LIN {X -44.717, Y 73.793, Z 53.25, A 0, B 90, C 0, E1 0, E2 0, E3 0, E4 0} C_DIS
LIN {X -42.585, Y 75.218, Z 53.25, A 0, B 90, C 0, E1 0, E2 0, E3 0, E4 0} C_DIS
LIN {X -40.331, Y 76.441, Z 53.25, A 0, B 90, C 0, E1 0, E2 0, E3 0, E4 0} C_DIS
LIN {X -37.99, Y 77.489, Z 53.25, A 0, B 90, C 0, E1 0, E2 0, E3 0, E4 0} C_DIS
LIN {X -35.582, Y 78.373, Z 53.25, A 0, B 90, C 0, E1 0, E2 0, E3 0, E4 0} C_DIS
LIN {X -33.121, Y 79.096, Z 53.25, A 0, B 90, C 0, E1 0, E2 0, E3 0, E4 0} C_DIS
LIN {X -30.62, Y 79.664, Z 53.25, A 0, B 90, C 0, E1 0, E2 0, E3 0, E4 0} C_DIS
LIN {X -28.088, Y 80.079, Z 53.25, A 0, B 90, C 0, E1 0, E2 0, E3 0, E4 0} C_DIS
LIN {X -25.538, Y 80.347, Z 53.25, A 0, B 90, C 0, E1 0, E2 0, E3 0, E4 0} C_DIS
LIN {X -22.976, Y 80.479, Z 53.25, A 0, B 90, C 0, E1 0, E2 0, E3 0, E4 0} C_DIS
LIN {X -20.411, Y 80.492, Z 53.25, A 0, B 90, C 0, E1 0, E2 0, E3 0, E4 0} C_DIS
LIN {X -17.847, Y 80.414, Z 53.25, A 0, B 90, C 0, E1 0, E2 0, E3 0, E4 0} C_DIS
LIN {X -15.284, Y 80.286, Z 53.25, A 0, B 90, C 0, E1 0, E2 0, E3 0, E4 0} C_DIS
LIN {X -12.723, Y 80.139, Z 53.25, A 0, B 90, C 0, E1 0, E2 0, E3 0, E4 0} C_DIS
LIN {X -10.163, Y 79.971, Z 53.25, A 0, B 90, C 0, E1 0, E2 0, E3 0, E4 0} C_DIS
LIN {X -7.607, Y 79.756, Z 53.25, A 0, B 90, C 0, E1 0, E2 0, E3 0, E4 0} C_DIS
LIN {X -5.057, Y 79.475, Z 53.25, A 0, B 90, C 0, E1 0, E2 0, E3 0, E4 0} C_DIS
LIN {X -2.517, Y 79.116, Z 53.25, A 0, B 90, C 0, E1 0, E2 0, E3 0, E4 0} C_DIS
LIN {X 0, Y 78.658, Z 53.25, A 0, B 90, C 0, E1 0, E2 0, E3 0, E4 0} C_DIS
LIN {X 2.44, Y 77.975, Z 53.25, A 0, B 90, C 0, E1 0, E2 0, E3 0, E4 0} C_DIS
LIN {X 4.923, Y 77.332, Z 53.25, A 0, B 90, C 0, E1 0, E2 0, E3 0, E4 0} C_DIS
LIN {X 7.38, Y 76.595, Z 53.25, A 0, B 90, C 0, E1 0, E2 0, E3 0, E4 0} C_DIS
LIN {X 9.8, Y 75.743, Z 53.25, A 0, B 90, C 0, E1 0, E2 0, E3 0, E4 0} C_DIS
LIN {X 12.156, Y 74.73, Z 53.25, A 0, B 90, C 0, E1 0, E2 0, E3 0, E4 0} C_DIS
LIN {X 14.414, Y 73.515, Z 53.25, A 0, B 90, C 0, E1 0, E2 0, E3 0, E4 0} C_DIS
LIN {X 16.599, Y 72.171, Z 53.25, A 0, B 90, C 0, E1 0, E2 0, E3 0, E4 0} C_DIS
LIN {X 18.763, Y 70.793, Z 53.25, A 0, B 90, C 0, E1 0, E2 0, E3 0, E4 0} C_DIS
LIN {X 20.937, Y 69.431, Z 53.25, A 0, B 90, C 0, E1 0, E2 0, E3 0, E4 0} C_DIS
LIN {X 23.139, Y 68.116, Z 53.25, A 0, B 90, C 0, E1 0, E2 0, E3 0, E4 0} C_DIS
LIN {X 25.379, Y 66.866, Z 53.25, A 0, B 90, C 0, E1 0, E2 0, E3 0, E4 0} C_DIS
LIN {X 27.66, Y 65.691, Z 53.25, A 0, B 90, C 0, E1 0, E2 0, E3 0, E4 0} C_DIS
LIN {X 29.977, Y 64.59, Z 53.25, A 0, B 90, C 0, E1 0, E2 0, E3 0, E4 0} C_DIS
LIN {X 32.325, Y 63.556, Z 53.25, A 0, B 90, C 0, E1 0, E2 0, E3 0, E4 0} C_DIS
LIN {X 34.697, Y 62.581, Z 53.25, A 0, B 90, C 0, E1 0, E2 0, E3 0, E4 0} C_DIS
LIN {X 37.093, Y 61.664, Z 53.25, A 0, B 90, C 0, E1 0, E2 0, E3 0, E4 0} C_DIS
LIN {X 39.514, Y 60.816, Z 53.25, A 0, B 90, C 0, E1 0, E2 0, E3 0, E4 0} C_DIS
LIN {X 41.962, Y 60.049, Z 53.25, A 0, B 90, C 0, E1 0, E2 0, E3 0, E4 0} C_DIS
LIN {X 44.431, Y 59.352, Z 53.25, A 0, B 90, C 0, E1 0, E2 0, E3 0, E4 0} C_DIS
LIN {X 46.908, Y 58.684, Z 53.25, A 0, B 90, C 0, E1 0, E2 0, E3 0, E4 0} C_DIS
LIN {X 49.381, Y 58.001, Z 53.25, A 0, B 90, C 0, E1 0, E2 0, E3 0, E4 0} C_DIS
LIN {X 51.841, Y 57.274, Z 53.25, A 0, B 90, C 0, E1 0, E2 0, E3 0, E4 0} C_DIS
LIN {X 54.281, Y 56.483, Z 53.25, A 0, B 90, C 0, E1 0, E2 0, E3 0, E4 0} C_DIS
LIN {X 56.696, Y 55.617, Z 53.25, A 0, B 90, C 0, E1 0, E2 0, E3 0, E4 0} C_DIS
LIN {X 59.079, Y 54.667, Z 53.25, A 0, B 90, C 0, E1 0, E2 0, E3 0, E4 0} C_DIS
LIN {X 61.423, Y 53.627, Z 53.25, A 0, B 90, C 0, E1 0, E2 0, E3 0, E4 0} C_DIS
LIN {X 63.722, Y 52.488, Z 53.25, A 0, B 90, C 0, E1 0, E2 0, E3 0, E4 0} C_DIS
LIN {X 65.964, Y 51.243, Z 53.25, A 0, B 90, C 0, E1 0, E2 0, E3 0, E4 0} C_DIS
LIN {X 68.135, Y 49.877, Z 53.25, A 0, B 90, C 0, E1 0, E2 0, E3 0, E4 0} C_DIS
LIN {X 70.208, Y 48.366, Z 53.25, A 0, B 90, C 0, E1 0, E2 0, E3 0, E4 0} C_DIS
LIN {X 72.121, Y 46.659, Z 53.25, A 0, B 90, C 0, E1 0, E2 0, E3 0, E4 0} C_DIS
LIN {X 73.793, Y 44.717, Z 53.25, A 0, B 90, C 0, E1 0, E2 0, E3 0, E4 0} C_DIS
LIN {X 75.218, Y 42.585, Z 53.25, A 0, B 90, C 0, E1 0, E2 0, E3 0, E4 0} C_DIS
LIN {X 76.441, Y 40.331, Z 53.25, A 0, B 90, C 0, E1 0, E2 0, E3 0, E4 0} C_DIS
LIN {X 77.489, Y 37.99, Z 53.25, A 0, B 90, C 0, E1 0, E2 0, E3 0, E4 0} C_DIS
LIN {X 78.373, Y 35.582, Z 53.25, A 0, B 90, C 0, E1 0, E2 0, E3 0, E4 0} C_DIS
LIN {X 79.096, Y 33.121, Z 53.25, A 0, B 90, C 0, E1 0, E2 0, E3 0, E4 0} C_DIS
LIN {X 79.664, Y 30.62, Z 53.25, A 0, B 90, C 0, E1 0, E2 0, E3 0, E4 0} C_DIS
LIN {X 80.079, Y 28.088, Z 53.25, A 0, B 90, C 0, E1 0, E2 0, E3 0, E4 0} C_DIS
LIN {X 80.347, Y 25.538, Z 53.25, A 0, B 90, C 0, E1 0, E2 0, E3 0, E4 0} C_DIS
LIN {X 80.479, Y 22.976, Z 53.25, A 0, B 90, C 0, E1 0, E2 0, E3 0, E4 0} C_DIS
LIN {X 80.492, Y 20.411, Z 53.25, A 0, B 90, C 0, E1 0, E2 0, E3 0, E4 0} C_DIS
LIN {X 80.414, Y 17.847, Z 53.25, A 0, B 90, C 0, E1 0, E2 0, E3 0, E4 0} C_DIS
LIN {X 80.286, Y 15.284, Z 53.25, A 0, B 90, C 0, E1 0, E2 0, E3 0, E4 0} C_DIS
LIN {X 80.139, Y 12.723, Z 53.25, A 0, B 90, C 0, E1 0, E2 0, E3 0, E4 0} C_DIS
LIN {X 79.971, Y 10.163, Z 53.25, A 0, B 90, C 0, E1 0, E2 0, E3 0, E4 0} C_DIS
LIN {X 79.756, Y 7.607, Z 53.25, A 0, B 90, C 0, E1 0, E2 0, E3 0, E4 0} C_DIS
LIN {X 79.475, Y 5.057, Z 53.25, A 0, B 90, C 0, E1 0, E2 0, E3 0, E4 0} C_DIS
LIN {X 79.116, Y 2.517, Z 53.25, A 0, B 90, C 0, E1 0, E2 0, E3 0, E4 0} C_DIS
LIN {X 78.658, Y 0, Z 53.25, A 0, B 90, C 0, E1 0, E2 0, E3 0, E4 0} C_DIS
LIN {X 77.975, Y -2.44, Z 53.25, A 0, B 90, C 0, E1 0, E2 0, E3 0, E4 0} C_DIS
LIN {X 77.332, Y -4.923, Z 53.25, A 0, B 90, C 0, E1 0, E2 0, E3 0, E4 0} C_DIS
LIN {X 76.595, Y -7.38, Z 53.25, A 0, B 90, C 0, E1 0, E2 0, E3 0, E4 0} C_DIS
LIN {X 75.743, Y -9.8, Z 53.25, A 0, B 90, C 0, E1 0, E2 0, E3 0, E4 0} C_DIS
LIN {X 74.73, Y -12.156, Z 53.25, A 0, B 90, C 0, E1 0, E2 0, E3 0, E4 0} C_DIS
LIN {X 73.515, Y -14.414, Z 53.25, A 0, B 90, C 0, E1 0, E2 0, E3 0, E4 0} C_DIS
LIN {X 72.171, Y -16.599, Z 53.25, A 0, B 90, C 0, E1 0, E2 0, E3 0, E4 0} C_DIS
LIN {X 70.793, Y -18.763, Z 53.25, A 0, B 90, C 0, E1 0, E2 0, E3 0, E4 0} C_DIS
LIN {X 69.431, Y -20.937, Z 53.25, A 0, B 90, C 0, E1 0, E2 0, E3 0, E4 0} C_DIS
LIN {X 68.116, Y -23.139, Z 53.25, A 0, B 90, C 0, E1 0, E2 0, E3 0, E4 0} C_DIS
LIN {X 66.866, Y -25.379, Z 53.25, A 0, B 90, C 0, E1 0, E2 0, E3 0, E4 0} C_DIS
LIN {X 65.691, Y -27.66, Z 53.25, A 0, B 90, C 0, E1 0, E2 0, E3 0, E4 0} C_DIS
LIN {X 64.59, Y -29.977, Z 53.25, A 0, B 90, C 0, E1 0, E2 0, E3 0, E4 0} C_DIS
LIN {X 63.556, Y -32.325, Z 53.25, A 0, B 90, C 0, E1 0, E2 0, E3 0, E4 0} C_DIS
LIN {X 62.581, Y -34.697, Z 53.25, A 0, B 90, C 0, E1 0, E2 0, E3 0, E4 0} C_DIS
LIN {X 61.664, Y -37.093, Z 53.25, A 0, B 90, C 0, E1 0, E2 0, E3 0, E4 0} C_DIS
LIN {X 60.816, Y -39.514, Z 53.25, A 0, B 90, C 0, E1 0, E2 0, E3 0, E4 0} C_DIS
LIN {X 60.049, Y -41.962, Z 53.25, A 0, B 90, C 0, E1 0, E2 0, E3 0, E4 0} C_DIS
LIN {X 59.352, Y -44.431, Z 53.25, A 0, B 90, C 0, E1 0, E2 0, E3 0, E4 0} C_DIS
LIN {X 58.684, Y -46.908, Z 53.25, A 0, B 90, C 0, E1 0, E2 0, E3 0, E4 0} C_DIS
LIN {X 58.001, Y -49.381, Z 53.25, A 0, B 90, C 0, E1 0, E2 0, E3 0, E4 0} C_DIS
LIN {X 57.274, Y -51.841, Z 53.25, A 0, B 90, C 0, E1 0, E2 0, E3 0, E4 0} C_DIS
LIN {X 56.483, Y -54.281, Z 53.25, A 0, B 90, C 0, E1 0, E2 0, E3 0, E4 0} C_DIS
LIN {X 55.617, Y -56.696, Z 53.25, A 0, B 90, C 0, E1 0, E2 0, E3 0, E4 0} C_DIS
LIN {X 54.667, Y -59.079, Z 53.25, A 0, B 90, C 0, E1 0, E2 0, E3 0, E4 0} C_DIS
LIN {X 53.627, Y -61.423, Z 53.25, A 0, B 90, C 0, E1 0, E2 0, E3 0, E4 0} C_DIS
LIN {X 52.488, Y -63.722, Z 53.25, A 0, B 90, C 0, E1 0, E2 0, E3 0, E4 0} C_DIS
LIN {X 51.243, Y -65.964, Z 53.25, A 0, B 90, C 0, E1 0, E2 0, E3 0, E4 0} C_DIS
LIN {X 49.877, Y -68.135, Z 53.25, A 0, B 90, C 0, E1 0, E2 0, E3 0, E4 0} C_DIS
LIN {X 48.366, Y -70.208, Z 53.25, A 0, B 90, C 0, E1 0, E2 0, E3 0, E4 0} C_DIS
LIN {X 46.659, Y -72.121, Z 53.25, A 0, B 90, C 0, E1 0, E2 0, E3 0, E4 0} C_DIS
LIN {X 44.717, Y -73.793, Z 53.25, A 0, B 90, C 0, E1 0, E2 0, E3 0, E4 0} C_DIS
LIN {X 42.585, Y -75.218, Z 53.25, A 0, B 90, C 0, E1 0, E2 0, E3 0, E4 0} C_DIS
LIN {X 40.331, Y -76.441, Z 53.25, A 0, B 90, C 0, E1 0, E2 0, E3 0, E4 0} C_DIS
LIN {X 37.99, Y -77.489, Z 53.25, A 0, B 90, C 0, E1 0, E2 0, E3 0, E4 0} C_DIS
LIN {X 35.582, Y -78.373, Z 53.25, A 0, B 90, C 0, E1 0, E2 0, E3 0, E4 0} C_DIS
LIN {X 33.121, Y -79.096, Z 53.25, A 0, B 90, C 0, E1 0, E2 0, E3 0, E4 0} C_DIS
LIN {X 30.62, Y -79.664, Z 53.25, A 0, B 90, C 0, E1 0, E2 0, E3 0, E4 0} C_DIS
LIN {X 28.088, Y -80.079, Z 53.25, A 0, B 90, C 0, E1 0, E2 0, E3 0, E4 0} C_DIS
LIN {X 25.538, Y -80.347, Z 53.25, A 0, B 90, C 0, E1 0, E2 0, E3 0, E4 0} C_DIS
LIN {X 22.976, Y -80.479, Z 53.25, A 0, B 90, C 0, E1 0, E2 0, E3 0, E4 0} C_DIS
LIN {X 20.411, Y -80.492, Z 53.25, A 0, B 90, C 0, E1 0, E2 0, E3 0, E4 0} C_DIS
LIN {X 17.847, Y -80.414, Z 53.25, A 0, B 90, C 0, E1 0, E2 0, E3 0, E4 0} C_DIS
LIN {X 15.284, Y -80.286, Z 53.25, A 0, B 90, C 0, E1 0, E2 0, E3 0, E4 0} C_DIS
LIN {X 12.723, Y -80.139, Z 53.25, A 0, B 90, C 0, E1 0, E2 0, E3 0, E4 0} C_DIS
LIN {X 10.163, Y -79.971, Z 53.25, A 0, B 90, C 0, E1 0, E2 0, E3 0, E4 0} C_DIS
LIN {X 7.607, Y -79.756, Z 53.25, A 0, B 90, C 0, E1 0, E2 0, E3 0, E4 0} C_DIS
LIN {X 5.057, Y -79.475, Z 53.25, A 0, B 90, C 0, E1 0, E2 0, E3 0, E4 0} C_DIS
LIN {X 2.517, Y -79.116, Z 53.25, A 0, B 90, C 0, E1 0, E2 0, E3 0, E4 0} C_DIS
LIN {X 0, Y -78.658, Z 53.25, A 0, B 90, C 0, E1 0, E2 0, E3 0, E4 0} C_DIS
LIN {X -2.44, Y -77.975, Z 53.25, A 0, B 90, C 0, E1 0, E2 0, E3 0, E4 0} C_DIS
LIN {X -4.923, Y -77.332, Z 53.25, A 0, B 90, C 0, E1 0, E2 0, E3 0, E4 0} C_DIS
LIN {X -7.38, Y -76.595, Z 53.25, A 0, B 90, C 0, E1 0, E2 0, E3 0, E4 0} C_DIS
LIN {X -9.8, Y -75.743, Z 53.25, A 0, B 90, C 0, E1 0, E2 0, E3 0, E4 0} C_DIS
LIN {X -12.156, Y -74.73, Z 53.25, A 0, B 90, C 0, E1 0, E2 0, E3 0, E4 0} C_DIS
LIN {X -14.414, Y -73.515, Z 53.25, A 0, B 90, C 0, E1 0, E2 0, E3 0, E4 0} C_DIS
LIN {X -16.599, Y -72.171, Z 53.25, A 0, B 90, C 0, E1 0, E2 0, E3 0, E4 0} C_DIS
LIN {X -18.763, Y -70.793, Z 53.25, A 0, B 90, C 0, E1 0, E2 0, E3 0, E4 0} C_DIS
LIN {X -20.937, Y -69.431, Z 53.25, A 0, B 90, C 0, E1 0, E2 0, E3 0, E4 0} C_DIS
LIN {X -23.139, Y -68.116, Z 53.25, A 0, B 90, C 0, E1 0, E2 0, E3 0, E4 0} C_DIS
LIN {X -25.379, Y -66.866, Z 53.25, A 0, B 90, C 0, E1 0, E2 0, E3 0, E4 0} C_DIS
LIN {X -27.66, Y -65.691, Z 53.25, A 0, B 90, C 0, E1 0, E2 0, E3 0, E4 0} C_DIS
LIN {X -29.977, Y -64.59, Z 53.25, A 0, B 90, C 0, E1 0, E2 0, E3 0, E4 0} C_DIS
LIN {X -32.325, Y -63.556, Z 53.25, A 0, B 90, C 0, E1 0, E2 0, E3 0, E4 0} C_DIS
LIN {X -34.697, Y -62.581, Z 53.25, A 0, B 90, C 0, E1 0, E2 0, E3 0, E4 0} C_DIS
LIN {X -37.093, Y -61.664, Z 53.25, A 0, B 90, C 0, E1 0, E2 0, E3 0, E4 0} C_DIS
LIN {X -39.514, Y -60.816, Z 53.25, A 0, B 90, C 0, E1 0, E2 0, E3 0, E4 0} C_DIS
LIN {X -41.962, Y -60.049, Z 53.25, A 0, B 90, C 0, E1 0, E2 0, E3 0, E4 0} C_DIS
LIN {X -44.431, Y -59.352, Z 53.25, A 0, B 90, C 0, E1 0, E2 0, E3 0, E4 0} C_DIS
LIN {X -46.908, Y -58.684, Z 53.25, A 0, B 90, C 0, E1 0, E2 0, E3 0, E4 0} C_DIS
LIN {X -49.381, Y -58.001, Z 53.25, A 0, B 90, C 0, E1 0, E2 0, E3 0, E4 0} C_DIS
LIN {X -51.841, Y -57.274, Z 53.25, A 0, B 90, C 0, E1 0, E2 0, E3 0, E4 0} C_DIS
LIN {X -54.281, Y -56.483, Z 53.25, A 0, B 90, C 0, E1 0, E2 0, E3 0, E4 0} C_DIS
LIN {X -56.696, Y -55.617, Z 53.25, A 0, B 90, C 0, E1 0, E2 0, E3 0, E4 0} C_DIS
LIN {X -59.079, Y -54.667, Z 53.25, A 0, B 90, C 0, E1 0, E2 0, E3 0, E4 0} C_DIS
LIN {X -61.423, Y -53.627, Z 53.25, A 0, B 90, C 0, E1 0, E2 0, E3 0, E4 0} C_DIS
LIN {X -63.722, Y -52.488, Z 53.25, A 0, B 90, C 0, E1 0, E2 0, E3 0, E4 0} C_DIS
LIN {X -65.964, Y -51.243, Z 53.25, A 0, B 90, C 0, E1 0, E2 0, E3 0, E4 0} C_DIS
LIN {X -68.135, Y -49.877, Z 53.25, A 0, B 90, C 0, E1 0, E2 0, E3 0, E4 0} C_DIS
LIN {X -70.208, Y -48.366, Z 53.25, A 0, B 90, C 0, E1 0, E2 0, E3 0, E4 0} C_DIS
LIN {X -72.121, Y -46.659, Z 53.25, A 0, B 90, C 0, E1 0, E2 0, E3 0, E4 0} C_DIS
LIN {X -73.793, Y -44.717, Z 53.25, A 0, B 90, C 0, E1 0, E2 0, E3 0, E4 0} C_DIS
LIN {X -75.218, Y -42.585, Z 53.25, A 0, B 90, C 0, E1 0, E2 0, E3 0, E4 0} C_DIS
LIN {X -76.441, Y -40.331, Z 53.25, A 0, B 90, C 0, E1 0, E2 0, E3 0, E4 0} C_DIS
LIN {X -77.489, Y -37.99, Z 53.25, A 0, B 90, C 0, E1 0, E2 0, E3 0, E4 0} C_DIS
LIN {X -78.373, Y -35.582, Z 53.25, A 0, B 90, C 0, E1 0, E2 0, E3 0, E4 0} C_DIS
LIN {X -79.096, Y -33.121, Z 53.25, A 0, B 90, C 0, E1 0, E2 0, E3 0, E4 0} C_DIS
LIN {X -79.664, Y -30.62, Z 53.25, A 0, B 90, C 0, E1 0, E2 0, E3 0, E4 0} C_DIS
LIN {X -80.079, Y -28.088, Z 53.25, A 0, B 90, C 0, E1 0, E2 0, E3 0, E4 0} C_DIS
LIN {X -80.347, Y -25.538, Z 53.25, A 0, B 90, C 0, E1 0, E2 0, E3 0, E4 0} C_DIS
LIN {X -80.479, Y -22.976, Z 53.25, A 0, B 90, C 0, E1 0, E2 0, E3 0, E4 0} C_DIS
LIN {X -80.492, Y -20.411, Z 53.25, A 0, B 90, C 0, E1 0, E2 0, E3 0, E4 0} C_DIS
LIN {X -80.414, Y -17.847, Z 53.25, A 0, B 90, C 0, E1 0, E2 0, E3 0, E4 0} C_DIS
LIN {X -80.286, Y -15.284, Z 53.25, A 0, B 90, C 0, E1 0, E2 0, E3 0, E4 0} C_DIS
LIN {X -80.139, Y -12.723, Z 53.25, A 0, B 90, C 0, E1 0, E2 0, E3 0, E4 0} C_DIS
LIN {X -79.971, Y -10.163, Z 53.25, A 0, B 90, C 0, E1 0, E2 0, E3 0, E4 0} C_DIS
LIN {X -79.756, Y -7.607, Z 53.25, A 0, B 90, C 0, E1 0, E2 0, E3 0, E4 0} C_DIS
LIN {X -79.475, Y -5.057, Z 53.25, A 0, B 90, C 0, E1 0, E2 0, E3 0, E4 0} C_DIS
LIN {X -79.116, Y -2.517, Z 53.25, A 0, B 90, C 0, E1 0, E2 0, E3 0, E4 0} C_DIS
LIN {X -78.665, Y 0, Z 55.75, A 0, B 90, C 0, E1 0, E2 0, E3 0, E4 0} C_DIS
LIN {X -77.946, Y 2.433, Z 55.75, A 0, B 90, C 0, E1 0, E2 0, E3 0, E4 0} C_DIS
LIN {X -77.272, Y 4.917, Z 55.75, A 0, B 90, C 0, E1 0, E2 0, E3 0, E4 0} C_DIS
LIN {X -76.503, Y 7.373, Z 55.75, A 0, B 90, C 0, E1 0, E2 0, E3 0, E4 0} C_DIS
LIN {X -75.619, Y 9.789, Z 55.75, A 0, B 90, C 0, E1 0, E2 0, E3 0, E4 0} C_DIS
LIN {X -74.571, Y 12.139, Z 55.75, A 0, B 90, C 0, E1 0, E2 0, E3 0, E4 0} C_DIS
LIN {X -73.32, Y 14.387, Z 55.75, A 0, B 90, C 0, E1 0, E2 0, E3 0, E4 0} C_DIS
LIN {X -71.942, Y 16.56, Z 55.75, A 0, B 90, C 0, E1 0, E2 0, E3 0, E4 0} C_DIS
LIN {X -70.532, Y 18.714, Z 55.75, A 0, B 90, C 0, E1 0, E2 0, E3 0, E4 0} C_DIS
LIN {X -69.142, Y 20.88, Z 55.75, A 0, B 90, C 0, E1 0, E2 0, E3 0, E4 0} C_DIS
LIN {X -67.803, Y 23.077, Z 55.75, A 0, B 90, C 0, E1 0, E2 0, E3 0, E4 0} C_DIS
LIN {X -66.534, Y 25.317, Z 55.75, A 0, B 90, C 0, E1 0, E2 0, E3 0, E4 0} C_DIS
LIN {X -65.347, Y 27.6, Z 55.75, A 0, B 90, C 0, E1 0, E2 0, E3 0, E4 0} C_DIS
LIN {X -64.241, Y 29.923, Z 55.75, A 0, B 90, C 0, E1 0, E2 0, E3 0, E4 0} C_DIS
LIN {X -63.207, Y 32.28, Z 55.75, A 0, B 90, C 0, E1 0, E2 0, E3 0, E4 0} C_DIS
LIN {X -62.239, Y 34.665, Z 55.75, A 0, B 90, C 0, E1 0, E2 0, E3 0, E4 0} C_DIS
LIN {X -61.336, Y 37.075, Z 55.75, A 0, B 90, C 0, E1 0, E2 0, E3 0, E4 0} C_DIS
LIN {X -60.509, Y 39.512, Z 55.75, A 0, B 90, C 0, E1 0, E2 0, E3 0, E4 0} C_DIS
LIN {X -59.769, Y 41.976, Z 55.75, A 0, B 90, C 0, E1 0, E2 0, E3 0, E4 0} C_DIS
LIN {X -59.105, Y 44.463, Z 55.75, A 0, B 90, C 0, E1 0, E2 0, E3 0, E4 0} C_DIS
LIN {X -58.473, Y 46.958, Z 55.75, A 0, B 90, C 0, E1 0, E2 0, E3 0, E4 0} C_DIS
LIN {X -57.827, Y 49.449, Z 55.75, A 0, B 90, C 0, E1 0, E2 0, E3 0, E4 0} C_DIS
LIN {X -57.137, Y 51.928, Z 55.75, A 0, B 90, C 0, E1 0, E2 0, E3 0, E4 0} C_DIS
LIN {X -56.382, Y 54.389, Z 55.75, A 0, B 90, C 0, E1 0, E2 0, E3 0, E4 0} C_DIS
LIN {X -55.552, Y 56.824, Z 55.75, A 0, B 90, C 0, E1 0, E2 0, E3 0, E4 0} C_DIS
LIN {X -54.636, Y 59.23, Z 55.75, A 0, B 90, C 0, E1 0, E2 0, E3 0, E4 0} C_DIS
LIN {X -53.628, Y 61.597, Z 55.75, A 0, B 90, C 0, E1 0, E2 0, E3 0, E4 0} C_DIS
LIN {X -52.52, Y 63.92, Z 55.75, A 0, B 90, C 0, E1 0, E2 0, E3 0, E4 0} C_DIS
LIN {X -51.303, Y 66.188, Z 55.75, A 0, B 90, C 0, E1 0, E2 0, E3 0, E4 0} C_DIS
LIN {X -49.964, Y 68.385, Z 55.75, A 0, B 90, C 0, E1 0, E2 0, E3 0, E4 0} C_DIS
LIN {X -48.475, Y 70.483, Z 55.75, A 0, B 90, C 0, E1 0, E2 0, E3 0, E4 0} C_DIS
LIN {X -46.785, Y 72.422, Z 55.75, A 0, B 90, C 0, E1 0, E2 0, E3 0, E4 0} C_DIS
LIN {X -44.848, Y 74.114, Z 55.75, A 0, B 90, C 0, E1 0, E2 0, E3 0, E4 0} C_DIS
LIN {X -42.715, Y 75.551, Z 55.75, A 0, B 90, C 0, E1 0, E2 0, E3 0, E4 0} C_DIS
LIN {X -40.455, Y 76.78, Z 55.75, A 0, B 90, C 0, E1 0, E2 0, E3 0, E4 0} C_DIS
LIN {X -38.105, Y 77.829, Z 55.75, A 0, B 90, C 0, E1 0, E2 0, E3 0, E4 0} C_DIS
LIN {X -35.687, Y 78.708, Z 55.75, A 0, B 90, C 0, E1 0, E2 0, E3 0, E4 0} C_DIS
LIN {X -33.215, Y 79.424, Z 55.75, A 0, B 90, C 0, E1 0, E2 0, E3 0, E4 0} C_DIS
LIN {X -30.703, Y 79.98, Z 55.75, A 0, B 90, C 0, E1 0, E2 0, E3 0, E4 0} C_DIS
LIN {X -28.161, Y 80.379, Z 55.75, A 0, B 90, C 0, E1 0, E2 0, E3 0, E4 0} C_DIS
LIN {X -25.599, Y 80.627, Z 55.75, A 0, B 90, C 0, E1 0, E2 0, E3 0, E4 0} C_DIS
LIN {X -23.028, Y 80.736, Z 55.75, A 0, B 90, C 0, E1 0, E2 0, E3 0, E4 0} C_DIS
LIN {X -20.455, Y 80.723, Z 55.75, A 0, B 90, C 0, E1 0, E2 0, E3 0, E4 0} C_DIS
LIN {X -17.884, Y 80.617, Z 55.75, A 0, B 90, C 0, E1 0, E2 0, E3 0, E4 0} C_DIS
LIN {X -15.315, Y 80.46, Z 55.75, A 0, B 90, C 0, E1 0, E2 0, E3 0, E4 0} C_DIS
LIN {X -12.747, Y 80.284, Z 55.75, A 0, B 90, C 0, E1 0, E2 0, E3 0, E4 0} C_DIS
LIN {X -10.181, Y 80.089, Z 55.75, A 0, B 90, C 0, E1 0, E2 0, E3 0, E4 0} C_DIS
LIN {X -7.619, Y 79.847, Z 55.75, A 0, B 90, C 0, E1 0, E2 0, E3 0, E4 0} C_DIS
LIN {X -5.064, Y 79.539, Z 55.75, A 0, B 90, C 0, E1 0, E2 0, E3 0, E4 0} C_DIS
LIN {X -2.52, Y 79.152, Z 55.75, A 0, B 90, C 0, E1 0, E2 0, E3 0, E4 0} C_DIS
LIN {X 0, Y 78.665, Z 55.75, A 0, B 90, C 0, E1 0, E2 0, E3 0, E4 0} C_DIS
LIN {X 2.433, Y 77.946, Z 55.75, A 0, B 90, C 0, E1 0, E2 0, E3 0, E4 0} C_DIS
LIN {X 4.917, Y 77.272, Z 55.75, A 0, B 90, C 0, E1 0, E2 0, E3 0, E4 0} C_DIS
LIN {X 7.373, Y 76.503, Z 55.75, A 0, B 90, C 0, E1 0, E2 0, E3 0, E4 0} C_DIS
LIN {X 9.789, Y 75.619, Z 55.75, A 0, B 90, C 0, E1 0, E2 0, E3 0, E4 0} C_DIS
LIN {X 12.139, Y 74.571, Z 55.75, A 0, B 90, C 0, E1 0, E2 0, E3 0, E4 0} C_DIS
LIN {X 14.387, Y 73.32, Z 55.75, A 0, B 90, C 0, E1 0, E2 0, E3 0, E4 0} C_DIS
LIN {X 16.56, Y 71.942, Z 55.75, A 0, B 90, C 0, E1 0, E2 0, E3 0, E4 0} C_DIS
LIN {X 18.714, Y 70.532, Z 55.75, A 0, B 90, C 0, E1 0, E2 0, E3 0, E4 0} C_DIS
LIN {X 20.88, Y 69.142, Z 55.75, A 0, B 90, C 0, E1 0, E2 0, E3 0, E4 0} C_DIS
LIN {X 23.077, Y 67.803, Z 55.75, A 0, B 90, C 0, E1 0, E2 0, E3 0, E4 0} C_DIS
LIN {X 25.317, Y 66.534, Z 55.75, A 0, B 90, C 0, E1 0, E2 0, E3 0, E4 0} C_DIS
LIN {X 27.6, Y 65.347, Z 55.75, A 0, B 90, C 0, E1 0, E2 0, E3 0, E4 0} C_DIS
LIN {X 29.923, Y 64.241, Z 55.75, A 0, B 90, C 0, E1 0, E2 0, E3 0, E4 0} C_DIS
LIN {X 32.28, Y 63.207, Z 55.75, A 0, B 90, C 0, E1 0, E2 0, E3 0, E4 0} C_DIS
LIN {X 34.665, Y 62.239, Z 55.75, A 0, B 90, C 0, E1 0, E2 0, E3 0, E4 0} C_DIS
LIN {X 37.075, Y 61.336, Z 55.75, A 0, B 90, C 0, E1 0, E2 0, E3 0, E4 0} C_DIS
LIN {X 39.512, Y 60.509, Z 55.75, A 0, B 90, C 0, E1 0, E2 0, E3 0, E4 0} C_DIS
LIN {X 41.976, Y 59.769, Z 55.75, A 0, B 90, C 0, E1 0, E2 0, E3 0, E4 0} C_DIS
LIN {X 44.463, Y 59.105, Z 55.75, A 0, B 90, C 0, E1 0, E2 0, E3 0, E4 0} C_DIS
LIN {X 46.958, Y 58.473, Z 55.75, A 0, B 90, C 0, E1 0, E2 0, E3 0, E4 0} C_DIS
LIN {X 49.449, Y 57.827, Z 55.75, A 0, B 90, C 0, E1 0, E2 0, E3 0, E4 0} C_DIS
LIN {X 51.928, Y 57.137, Z 55.75, A 0, B 90, C 0, E1 0, E2 0, E3 0, E4 0} C_DIS
LIN {X 54.389, Y 56.382, Z 55.75, A 0, B 90, C 0, E1 0, E2 0, E3 0, E4 0} C_DIS
LIN {X 56.824, Y 55.552, Z 55.75, A 0, B 90, C 0, E1 0, E2 0, E3 0, E4 0} C_DIS
LIN {X 59.23, Y 54.636, Z 55.75, A 0, B 90, C 0, E1 0, E2 0, E3 0, E4 0} C_DIS
LIN {X 61.597, Y 53.628, Z 55.75, A 0, B 90, C 0, E1 0, E2 0, E3 0, E4 0} C_DIS
LIN {X 63.92, Y 52.52, Z 55.75, A 0, B 90, C 0, E1 0, E2 0, E3 0, E4 0} C_DIS
LIN {X 66.188, Y 51.303, Z 55.75, A 0, B 90, C 0, E1 0, E2 0, E3 0, E4 0} C_DIS
LIN {X 68.385, Y 49.964, Z 55.75, A 0, B 90, C 0, E1 0, E2 0, E3 0, E4 0} C_DIS
LIN {X 70.483, Y 48.475, Z 55.75, A 0, B 90, C 0, E1 0, E2 0, E3 0, E4 0} C_DIS
LIN {X 72.422, Y 46.785, Z 55.75, A 0, B 90, C 0, E1 0, E2 0, E3 0, E4 0} C_DIS
LIN {X 74.114, Y 44.848, Z 55.75, A 0, B 90, C 0, E1 0, E2 0, E3 0, E4 0} C_DIS
LIN {X 75.551, Y 42.715, Z 55.75, A 0, B 90, C 0, E1 0, E2 0, E3 0, E4 0} C_DIS
LIN {X 76.78, Y 40.455, Z 55.75, A 0, B 90, C 0, E1 0, E2 0, E3 0, E4 0} C_DIS
LIN {X 77.829, Y 38.105, Z 55.75, A 0, B 90, C 0, E1 0, E2 0, E3 0, E4 0} C_DIS
LIN {X 78.708, Y 35.687, Z 55.75, A 0, B 90, C 0, E1 0, E2 0, E3 0, E4 0} C_DIS
LIN {X 79.424, Y 33.215, Z 55.75, A 0, B 90, C 0, E1 0, E2 0, E3 0, E4 0} C_DIS
LIN {X 79.98, Y 30.703, Z 55.75, A 0, B 90, C 0, E1 0, E2 0, E3 0, E4 0} C_DIS
LIN {X 80.379, Y 28.161, Z 55.75, A 0, B 90, C 0, E1 0, E2 0, E3 0, E4 0} C_DIS
LIN {X 80.627, Y 25.599, Z 55.75, A 0, B 90, C 0, E1 0, E2 0, E3 0, E4 0} C_DIS
LIN {X 80.736, Y 23.028, Z 55.75, A 0, B 90, C 0, E1 0, E2 0, E3 0, E4 0} C_DIS
LIN {X 80.723, Y 20.455, Z 55.75, A 0, B 90, C 0, E1 0, E2 0, E3 0, E4 0} C_DIS
LIN {X 80.617, Y 17.884, Z 55.75, A 0, B 90, C 0, E1 0, E2 0, E3 0, E4 0} C_DIS
LIN {X 80.46, Y 15.315, Z 55.75, A 0, B 90, C 0, E1 0, E2 0, E3 0, E4 0} C_DIS
LIN {X 80.284, Y 12.747, Z 55.75, A 0, B 90, C 0, E1 0, E2 0, E3 0, E4 0} C_DIS
LIN {X 80.089, Y 10.181, Z 55.75, A 0, B 90, C 0, E1 0, E2 0, E3 0, E4 0} C_DIS
LIN {X 79.847, Y 7.619, Z 55.75, A 0, B 90, C 0, E1 0, E2 0, E3 0, E4 0} C_DIS
LIN {X 79.539, Y 5.064, Z 55.75, A 0, B 90, C 0, E1 0, E2 0, E3 0, E4 0} C_DIS
LIN {X 79.152, Y 2.52, Z 55.75, A 0, B 90, C 0, E1 0, E2 0, E3 0, E4 0} C_DIS
LIN {X 78.665, Y 0, Z 55.75, A 0, B 90, C 0, E1 0, E2 0, E3 0, E4 0} C_DIS
LIN {X 77.946, Y -2.433, Z 55.75, A 0, B 90, C 0, E1 0, E2 0, E3 0, E4 0} C_DIS
LIN {X 77.272, Y -4.917, Z 55.75, A 0, B 90, C 0, E1 0, E2 0, E3 0, E4 0} C_DIS
LIN {X 76.503, Y -7.373, Z 55.75, A 0, B 90, C 0, E1 0, E2 0, E3 0, E4 0} C_DIS
LIN {X 75.619, Y -9.789, Z 55.75, A 0, B 90, C 0, E1 0, E2 0, E3 0, E4 0} C_DIS
LIN {X 74.571, Y -12.139, Z 55.75, A 0, B 90, C 0, E1 0, E2 0, E3 0, E4 0} C_DIS
LIN {X 73.32, Y -14.387, Z 55.75, A 0, B 90, C 0, E1 0, E2 0, E3 0, E4 0} C_DIS
LIN {X 71.942, Y -16.56, Z 55.75, A 0, B 90, C 0, E1 0, E2 0, E3 0, E4 0} C_DIS
LIN {X 70.532, Y -18.714, Z 55.75, A 0, B 90, C 0, E1 0, E2 0, E3 0, E4 0} C_DIS
LIN {X 69.142, Y -20.88, Z 55.75, A 0, B 90, C 0, E1 0, E2 0, E3 0, E4 0} C_DIS
LIN {X 67.803, Y -23.077, Z 55.75, A 0, B 90, C 0, E1 0, E2 0, E3 0, E4 0} C_DIS
LIN {X 66.534, Y -25.317, Z 55.75, A 0, B 90, C 0, E1 0, E2 0, E3 0, E4 0} C_DIS
LIN {X 65.347, Y -27.6, Z 55.75, A 0, B 90, C 0, E1 0, E2 0, E3 0, E4 0} C_DIS
LIN {X 64.241, Y -29.923, Z 55.75, A 0, B 90, C 0, E1 0, E2 0, E3 0, E4 0} C_DIS
LIN {X 63.207, Y -32.28, Z 55.75, A 0, B 90, C 0, E1 0, E2 0, E3 0, E4 0} C_DIS
LIN {X 62.239, Y -34.665, Z 55.75, A 0, B 90, C 0, E1 0, E2 0, E3 0, E4 0} C_DIS
LIN {X 61.336, Y -37.075, Z 55.75, A 0, B 90, C 0, E1 0, E2 0, E3 0, E4 0} C_DIS
LIN {X 60.509, Y -39.512, Z 55.75, A 0, B 90, C 0, E1 0, E2 0, E3 0, E4 0} C_DIS
LIN {X 59.769, Y -41.976, Z 55.75, A 0, B 90, C 0, E1 0, E2 0, E3 0, E4 0} C_DIS
LIN {X 59.105, Y -44.463, Z 55.75, A 0, B 90, C 0, E1 0, E2 0, E3 0, E4 0} C_DIS
LIN {X 58.473, Y -46.958, Z 55.75, A 0, B 90, C 0, E1 0, E2 0, E3 0, E4 0} C_DIS
LIN {X 57.827, Y -49.449, Z 55.75, A 0, B 90, C 0, E1 0, E2 0, E3 0, E4 0} C_DIS
LIN {X 57.137, Y -51.928, Z 55.75, A 0, B 90, C 0, E1 0, E2 0, E3 0, E4 0} C_DIS
LIN {X 56.382, Y -54.389, Z 55.75, A 0, B 90, C 0, E1 0, E2 0, E3 0, E4 0} C_DIS
LIN {X 55.552, Y -56.824, Z 55.75, A 0, B 90, C 0, E1 0, E2 0, E3 0, E4 0} C_DIS
LIN {X 54.636, Y -59.23, Z 55.75, A 0, B 90, C 0, E1 0, E2 0, E3 0, E4 0} C_DIS
LIN {X 53.628, Y -61.597, Z 55.75, A 0, B 90, C 0, E1 0, E2 0, E3 0, E4 0} C_DIS
LIN {X 52.52, Y -63.92, Z 55.75, A 0, B 90, C 0, E1 0, E2 0, E3 0, E4 0} C_DIS
LIN {X 51.303, Y -66.188, Z 55.75, A 0, B 90, C 0, E1 0, E2 0, E3 0, E4 0} C_DIS
LIN {X 49.964, Y -68.385, Z 55.75, A 0, B 90, C 0, E1 0, E2 0, E3 0, E4 0} C_DIS
LIN {X 48.475, Y -70.483, Z 55.75, A 0, B 90, C 0, E1 0, E2 0, E3 0, E4 0} C_DIS
LIN {X 46.785, Y -72.422, Z 55.75, A 0, B 90, C 0, E1 0, E2 0, E3 0, E4 0} C_DIS
LIN {X 44.848, Y -74.114, Z 55.75, A 0, B 90, C 0, E1 0, E2 0, E3 0, E4 0} C_DIS
LIN {X 42.715, Y -75.551, Z 55.75, A 0, B 90, C 0, E1 0, E2 0, E3 0, E4 0} C_DIS
LIN {X 40.455, Y -76.78, Z 55.75, A 0, B 90, C 0, E1 0, E2 0, E3 0, E4 0} C_DIS
LIN {X 38.105, Y -77.829, Z 55.75, A 0, B 90, C 0, E1 0, E2 0, E3 0, E4 0} C_DIS
LIN {X 35.687, Y -78.708, Z 55.75, A 0, B 90, C 0, E1 0, E2 0, E3 0, E4 0} C_DIS
LIN {X 33.215, Y -79.424, Z 55.75, A 0, B 90, C 0, E1 0, E2 0, E3 0, E4 0} C_DIS
LIN {X 30.703, Y -79.98, Z 55.75, A 0, B 90, C 0, E1 0, E2 0, E3 0, E4 0} C_DIS
LIN {X 28.161, Y -80.379, Z 55.75, A 0, B 90, C 0, E1 0, E2 0, E3 0, E4 0} C_DIS
LIN {X 25.599, Y -80.627, Z 55.75, A 0, B 90, C 0, E1 0, E2 0, E3 0, E4 0} C_DIS
LIN {X 23.028, Y -80.736, Z 55.75, A 0, B 90, C 0, E1 0, E2 0, E3 0, E4 0} C_DIS
LIN {X 20.455, Y -80.723, Z 55.75, A 0, B 90, C 0, E1 0, E2 0, E3 0, E4 0} C_DIS
LIN {X 17.884, Y -80.617, Z 55.75, A 0, B 90, C 0, E1 0, E2 0, E3 0, E4 0} C_DIS
LIN {X 15.315, Y -80.46, Z 55.75, A 0, B 90, C 0, E1 0, E2 0, E3 0, E4 0} C_DIS
LIN {X 12.747, Y -80.284, Z 55.75, A 0, B 90, C 0, E1 0, E2 0, E3 0, E4 0} C_DIS
LIN {X 10.181, Y -80.089, Z 55.75, A 0, B 90, C 0, E1 0, E2 0, E3 0, E4 0} C_DIS
LIN {X 7.619, Y -79.847, Z 55.75, A 0, B 90, C 0, E1 0, E2 0, E3 0, E4 0} C_DIS
LIN {X 5.064, Y -79.539, Z 55.75, A 0, B 90, C 0, E1 0, E2 0, E3 0, E4 0} C_DIS
LIN {X 2.52, Y -79.152, Z 55.75, A 0, B 90, C 0, E1 0, E2 0, E3 0, E4 0} C_DIS
LIN {X 0, Y -78.665, Z 55.75, A 0, B 90, C 0, E1 0, E2 0, E3 0, E4 0} C_DIS
LIN {X -2.433, Y -77.946, Z 55.75, A 0, B 90, C 0, E1 0, E2 0, E3 0, E4 0} C_DIS
LIN {X -4.917, Y -77.272, Z 55.75, A 0, B 90, C 0, E1 0, E2 0, E3 0, E4 0} C_DIS
LIN {X -7.373, Y -76.503, Z 55.75, A 0, B 90, C 0, E1 0, E2 0, E3 0, E4 0} C_DIS
LIN {X -9.789, Y -75.619, Z 55.75, A 0, B 90, C 0, E1 0, E2 0, E3 0, E4 0} C_DIS
LIN {X -12.139, Y -74.571, Z 55.75, A 0, B 90, C 0, E1 0, E2 0, E3 0, E4 0} C_DIS
LIN {X -14.387, Y -73.32, Z 55.75, A 0, B 90, C 0, E1 0, E2 0, E3 0, E4 0} C_DIS
LIN {X -16.56, Y -71.942, Z 55.75, A 0, B 90, C 0, E1 0, E2 0, E3 0, E4 0} C_DIS
LIN {X -18.714, Y -70.532, Z 55.75, A 0, B 90, C 0, E1 0, E2 0, E3 0, E4 0} C_DIS
LIN {X -20.88, Y -69.142, Z 55.75, A 0, B 90, C 0, E1 0, E2 0, E3 0, E4 0} C_DIS
LIN {X -23.077, Y -67.803, Z 55.75, A 0, B 90, C 0, E1 0, E2 0, E3 0, E4 0} C_DIS
LIN {X -25.317, Y -66.534, Z 55.75, A 0, B 90, C 0, E1 0, E2 0, E3 0, E4 0} C_DIS
LIN {X -27.6, Y -65.347, Z 55.75, A 0, B 90, C 0, E1 0, E2 0, E3 0, E4 0} C_DIS
LIN {X -29.923, Y -64.241, Z 55.75, A 0, B 90, C 0, E1 0, E2 0, E3 0, E4 0} C_DIS
LIN {X -32.28, Y -63.207, Z 55.75, A 0, B 90, C 0, E1 0, E2 0, E3 0, E4 0} C_DIS
LIN {X -34.665, Y -62.239, Z 55.75, A 0, B 90, C 0, E1 0, E2 0, E3 0, E4 0} C_DIS
LIN {X -37.075, Y -61.336, Z 55.75, A 0, B 90, C 0, E1 0, E2 0, E3 0, E4 0} C_DIS
LIN {X -39.512, Y -60.509, Z 55.75, A 0, B 90, C 0, E1 0, E2 0, E3 0, E4 0} C_DIS
LIN {X -41.976, Y -59.769, Z 55.75, A 0, B 90, C 0, E1 0, E2 0, E3 0, E4 0} C_DIS
LIN {X -44.463, Y -59.105, Z 55.75, A 0, B 90, C 0, E1 0, E2 0, E3 0, E4 0} C_DIS
LIN {X -46.958, Y -58.473, Z 55.75, A 0, B 90, C 0, E1 0, E2 0, E3 0, E4 0} C_DIS
LIN {X -49.449, Y -57.827, Z 55.75, A 0, B 90, C 0, E1 0, E2 0, E3 0, E4 0} C_DIS
LIN {X -51.928, Y -57.137, Z 55.75, A 0, B 90, C 0, E1 0, E2 0, E3 0, E4 0} C_DIS
LIN {X -54.389, Y -56.382, Z 55.75, A 0, B 90, C 0, E1 0, E2 0, E3 0, E4 0} C_DIS
LIN {X -56.824, Y -55.552, Z 55.75, A 0, B 90, C 0, E1 0, E2 0, E3 0, E4 0} C_DIS
LIN {X -59.23, Y -54.636, Z 55.75, A 0, B 90, C 0, E1 0, E2 0, E3 0, E4 0} C_DIS
LIN {X -61.597, Y -53.628, Z 55.75, A 0, B 90, C 0, E1 0, E2 0, E3 0, E4 0} C_DIS
LIN {X -63.92, Y -52.52, Z 55.75, A 0, B 90, C 0, E1 0, E2 0, E3 0, E4 0} C_DIS
LIN {X -66.188, Y -51.303, Z 55.75, A 0, B 90, C 0, E1 0, E2 0, E3 0, E4 0} C_DIS
LIN {X -68.385, Y -49.964, Z 55.75, A 0, B 90, C 0, E1 0, E2 0, E3 0, E4 0} C_DIS
LIN {X -70.483, Y -48.475, Z 55.75, A 0, B 90, C 0, E1 0, E2 0, E3 0, E4 0} C_DIS
LIN {X -72.422, Y -46.785, Z 55.75, A 0, B 90, C 0, E1 0, E2 0, E3 0, E4 0} C_DIS
LIN {X -74.114, Y -44.848, Z 55.75, A 0, B 90, C 0, E1 0, E2 0, E3 0, E4 0} C_DIS
LIN {X -75.551, Y -42.715, Z 55.75, A 0, B 90, C 0, E1 0, E2 0, E3 0, E4 0} C_DIS
LIN {X -76.78, Y -40.455, Z 55.75, A 0, B 90, C 0, E1 0, E2 0, E3 0, E4 0} C_DIS
LIN {X -77.829, Y -38.105, Z 55.75, A 0, B 90, C 0, E1 0, E2 0, E3 0, E4 0} C_DIS
LIN {X -78.708, Y -35.687, Z 55.75, A 0, B 90, C 0, E1 0, E2 0, E3 0, E4 0} C_DIS
LIN {X -79.424, Y -33.215, Z 55.75, A 0, B 90, C 0, E1 0, E2 0, E3 0, E4 0} C_DIS
LIN {X -79.98, Y -30.703, Z 55.75, A 0, B 90, C 0, E1 0, E2 0, E3 0, E4 0} C_DIS
LIN {X -80.379, Y -28.161, Z 55.75, A 0, B 90, C 0, E1 0, E2 0, E3 0, E4 0} C_DIS
LIN {X -80.627, Y -25.599, Z 55.75, A 0, B 90, C 0, E1 0, E2 0, E3 0, E4 0} C_DIS
LIN {X -80.736, Y -23.028, Z 55.75, A 0, B 90, C 0, E1 0, E2 0, E3 0, E4 0} C_DIS
LIN {X -80.723, Y -20.455, Z 55.75, A 0, B 90, C 0, E1 0, E2 0, E3 0, E4 0} C_DIS
LIN {X -80.617, Y -17.884, Z 55.75, A 0, B 90, C 0, E1 0, E2 0, E3 0, E4 0} C_DIS
LIN {X -80.46, Y -15.315, Z 55.75, A 0, B 90, C 0, E1 0, E2 0, E3 0, E4 0} C_DIS
LIN {X -80.284, Y -12.747, Z 55.75, A 0, B 90, C 0, E1 0, E2 0, E3 0, E4 0} C_DIS
LIN {X -80.089, Y -10.181, Z 55.75, A 0, B 90, C 0, E1 0, E2 0, E3 0, E4 0} C_DIS
LIN {X -79.847, Y -7.619, Z 55.75, A 0, B 90, C 0, E1 0, E2 0, E3 0, E4 0} C_DIS
LIN {X -79.539, Y -5.064, Z 55.75, A 0, B 90, C 0, E1 0, E2 0, E3 0, E4 0} C_DIS
LIN {X -79.152, Y -2.52, Z 55.75, A 0, B 90, C 0, E1 0, E2 0, E3 0, E4 0} C_DIS
LIN {X -78.682, Y 0, Z 58.25, A 0, B 90, C 0, E1 0, E2 0, E3 0, E4 0} C_DIS
LIN {X -77.926, Y 2.426, Z 58.25, A 0, B 90, C 0, E1 0, E2 0, E3 0, E4 0} C_DIS
LIN {X -77.221, Y 4.91, Z 58.25, A 0, B 90, C 0, E1 0, E2 0, E3 0, E4 0} C_DIS
LIN {X -76.421, Y 7.365, Z 58.25, A 0, B 90, C 0, E1 0, E2 0, E3 0, E4 0} C_DIS
LIN {X -75.505, Y 9.779, Z 58.25, A 0, B 90, C 0, E1 0, E2 0, E3 0, E4 0} C_DIS
LIN {X -74.423, Y 12.123, Z 58.25, A 0, B 90, C 0, E1 0, E2 0, E3 0, E4 0} C_DIS
LIN {X -73.137, Y 14.361, Z 58.25, A 0, B 90, C 0, E1 0, E2 0, E3 0, E4 0} C_DIS
LIN {X -71.725, Y 16.523, Z 58.25, A 0, B 90, C 0, E1 0, E2 0, E3 0, E4 0} C_DIS
LIN {X -70.284, Y 18.666, Z 58.25, A 0, B 90, C 0, E1 0, E2 0, E3 0, E4 0} C_DIS
LIN {X -68.867, Y 20.824, Z 58.25, A 0, B 90, C 0, E1 0, E2 0, E3 0, E4 0} C_DIS
LIN {X -67.505, Y 23.018, Z 58.25, A 0, B 90, C 0, E1 0, E2 0, E3 0, E4 0} C_DIS
LIN {X -66.22, Y 25.257, Z 58.25, A 0, B 90, C 0, E1 0, E2 0, E3 0, E4 0} C_DIS
LIN {X -65.021, Y 27.544, Z 58.25, A 0, B 90, C 0, E1 0, E2 0, E3 0, E4 0} C_DIS
LIN {X -63.909, Y 29.875, Z 58.25, A 0, B 90, C 0, E1 0, E2 0, E3 0, E4 0} C_DIS
LIN {X -62.876, Y 32.241, Z 58.25, A 0, B 90, C 0, E1 0, E2 0, E3 0, E4 0} C_DIS
LIN {X -61.915, Y 34.638, Z 58.25, A 0, B 90, C 0, E1 0, E2 0, E3 0, E4 0} C_DIS
LIN {X -61.026, Y 37.062, Z 58.25, A 0, B 90, C 0, E1 0, E2 0, E3 0, E4 0} C_DIS
LIN {X -60.218, Y 39.515, Z 58.25, A 0, B 90, C 0, E1 0, E2 0, E3 0, E4 0} C_DIS
LIN {X -59.506, Y 41.997, Z 58.25, A 0, B 90, C 0, E1 0, E2 0, E3 0, E4 0} C_DIS
LIN {X -58.874, Y 44.5, Z 58.25, A 0, B 90, C 0, E1 0, E2 0, E3 0, E4 0} C_DIS
LIN {X -58.277, Y 47.013, Z 58.25, A 0, B 90, C 0, E1 0, E2 0, E3 0, E4 0} C_DIS
LIN {X -57.666, Y 49.522, Z 58.25, A 0, B 90, C 0, E1 0, E2 0, E3 0, E4 0} C_DIS
LIN {X -57.011, Y 52.019, Z 58.25, A 0, B 90, C 0, E1 0, E2 0, E3 0, E4 0} C_DIS
LIN {X -56.292, Y 54.499, Z 58.25, A 0, B 90, C 0, E1 0, E2 0, E3 0, E4 0} C_DIS
LIN {X -55.495, Y 56.955, Z 58.25, A 0, B 90, C 0, E1 0, E2 0, E3 0, E4 0} C_DIS
LIN {X -54.612, Y 59.382, Z 58.25, A 0, B 90, C 0, E1 0, E2 0, E3 0, E4 0} C_DIS
LIN {X -53.635, Y 61.772, Z 58.25, A 0, B 90, C 0, E1 0, E2 0, E3 0, E4 0} C_DIS
LIN {X -52.557, Y 64.118, Z 58.25, A 0, B 90, C 0, E1 0, E2 0, E3 0, E4 0} C_DIS
LIN {X -51.368, Y 66.41, Z 58.25, A 0, B 90, C 0, E1 0, E2 0, E3 0, E4 0} C_DIS
LIN {X -50.053, Y 68.632, Z 58.25, A 0, B 90, C 0, E1 0, E2 0, E3 0, E4 0} C_DIS
LIN {X -48.586, Y 70.756, Z 58.25, A 0, B 90, C 0, E1 0, E2 0, E3 0, E4 0} C_DIS
LIN {X -46.911, Y 72.719, Z 58.25, A 0, B 90, C 0, E1 0, E2 0, E3 0, E4 0} C_DIS
LIN {X -44.981, Y 74.431, Z 58.25, A 0, B 90, C 0, E1 0, E2 0, E3 0, E4 0} C_DIS
LIN {X -42.846, Y 75.881, Z 58.25, A 0, B 90, C 0, E1 0, E2 0, E3 0, E4 0} C_DIS
LIN {X -40.58, Y 77.117, Z 58.25, A 0, B 90, C 0, E1 0, E2 0, E3 0, E4 0} C_DIS
LIN {X -38.221, Y 78.167, Z 58.25, A 0, B 90, C 0, E1 0, E2 0, E3 0, E4 0} C_DIS
LIN {X -35.793, Y 79.044, Z 58.25, A 0, B 90, C 0, E1 0, E2 0, E3 0, E4 0} C_DIS
LIN {X -33.311, Y 79.753, Z 58.25, A 0, B 90, C 0, E1 0, E2 0, E3 0, E4 0} C_DIS
LIN {X -30.787, Y 80.297, Z 58.25, A 0, B 90, C 0, E1 0, E2 0, E3 0, E4 0} C_DIS
LIN {X -28.234, Y 80.681, Z 58.25, A 0, B 90, C 0, E1 0, E2 0, E3 0, E4 0} C_DIS
LIN {X -25.662, Y 80.911, Z 58.25, A 0, B 90, C 0, E1 0, E2 0, E3 0, E4 0} C_DIS
LIN {X -23.082, Y 80.999, Z 58.25, A 0, B 90, C 0, E1 0, E2 0, E3 0, E4 0} C_DIS
LIN {X -20.5, Y 80.961, Z 58.25, A 0, B 90, C 0, E1 0, E2 0, E3 0, E4 0} C_DIS
LIN {X -17.921, Y 80.827, Z 58.25, A 0, B 90, C 0, E1 0, E2 0, E3 0, E4 0} C_DIS
LIN {X -15.346, Y 80.642, Z 58.25, A 0, B 90, C 0, E1 0, E2 0, E3 0, E4 0} C_DIS
LIN {X -12.771, Y 80.439, Z 58.25, A 0, B 90, C 0, E1 0, E2 0, E3 0, E4 0} C_DIS
LIN {X -10.199, Y 80.216, Z 58.25, A 0, B 90, C 0, E1 0, E2 0, E3 0, E4 0} C_DIS
LIN {X -7.631, Y 79.947, Z 58.25, A 0, B 90, C 0, E1 0, E2 0, E3 0, E4 0} C_DIS
LIN {X -5.07, Y 79.611, Z 58.25, A 0, B 90, C 0, E1 0, E2 0, E3 0, E4 0} C_DIS
LIN {X -2.522, Y 79.197, Z 58.25, A 0, B 90, C 0, E1 0, E2 0, E3 0, E4 0} C_DIS
LIN {X 0, Y 78.682, Z 58.25, A 0, B 90, C 0, E1 0, E2 0, E3 0, E4 0} C_DIS
LIN {X 2.426, Y 77.926, Z 58.25, A 0, B 90, C 0, E1 0, E2 0, E3 0, E4 0} C_DIS
LIN {X 4.91, Y 77.221, Z 58.25, A 0, B 90, C 0, E1 0, E2 0, E3 0, E4 0} C_DIS
LIN {X 7.365, Y 76.421, Z 58.25, A 0, B 90, C 0, E1 0, E2 0, E3 0, E4 0} C_DIS
LIN {X 9.779, Y 75.505, Z 58.25, A 0, B 90, C 0, E1 0, E2 0, E3 0, E4 0} C_DIS
LIN {X 12.123, Y 74.423, Z 58.25, A 0, B 90, C 0, E1 0, E2 0, E3 0, E4 0} C_DIS
LIN {X 14.361, Y 73.137, Z 58.25, A 0, B 90, C 0, E1 0, E2 0, E3 0, E4 0} C_DIS
LIN {X 16.523, Y 71.725, Z 58.25, A 0, B 90, C 0, E1 0, E2 0, E3 0, E4 0} C_DIS
LIN {X 18.666, Y 70.284, Z 58.25, A 0, B 90, C 0, E1 0, E2 0, E3 0, E4 0} C_DIS
LIN {X 20.824, Y 68.867, Z 58.25, A 0, B 90, C 0, E1 0, E2 0, E3 0, E4 0} C_DIS
LIN {X 23.018, Y 67.505, Z 58.25, A 0, B 90, C 0, E1 0, E2 0, E3 0, E4 0} C_DIS
LIN {X 25.257, Y 66.22, Z 58.25, A 0, B 90, C 0, E1 0, E2 0, E3 0, E4 0} C_DIS
LIN {X 27.544, Y 65.021, Z 58.25, A 0, B 90, C 0, E1 0, E2 0, E3 0, E4 0} C_DIS
LIN {X 29.875, Y 63.909, Z 58.25, A 0, B 90, C 0, E1 0, E2 0, E3 0, E4 0} C_DIS
LIN {X 32.241, Y 62.876, Z 58.25, A 0, B 90, C 0, E1 0, E2 0, E3 0, E4 0} C_DIS
LIN {X 34.638, Y 61.915, Z 58.25, A 0, B 90, C 0, E1 0, E2 0, E3 0, E4 0} C_DIS
LIN {X 37.062, Y 61.026, Z 58.25, A 0, B 90, C 0, E1 0, E2 0, E3 0, E4 0} C_DIS
LIN {X 39.515, Y 60.218, Z 58.25, A 0, B 90, C 0, E1 0, E2 0, E3 0, E4 0} C_DIS
LIN {X 41.997, Y 59.506, Z 58.25, A 0, B 90, C 0, E1 0, E2 0, E3 0, E4 0} C_DIS
LIN {X 44.5, Y 58.874, Z 58.25, A 0, B 90, C 0, E1 0, E2 0, E3 0, E4 0} C_DIS
LIN {X 47.013, Y 58.277, Z 58.25, A 0, B 90, C 0, E1 0, E2 0, E3 0, E4 0} C_DIS
LIN {X 49.522, Y 57.666, Z 58.25, A 0, B 90, C 0, E1 0, E2 0, E3 0, E4 0} C_DIS
LIN {X 52.019, Y 57.011, Z 58.25, A 0, B 90, C 0, E1 0, E2 0, E3 0, E4 0} C_DIS
LIN {X 54.499, Y 56.292, Z 58.25, A 0, B 90, C 0, E1 0, E2 0, E3 0, E4 0} C_DIS
LIN {X 56.955, Y 55.495, Z 58.25, A 0, B 90, C 0, E1 0, E2 0, E3 0, E4 0} C_DIS
LIN {X 59.382, Y 54.612, Z 58.25, A 0, B 90, C 0, E1 0, E2 0, E3 0, E4 0} C_DIS
LIN {X 61.772, Y 53.635, Z 58.25, A 0, B 90, C 0, E1 0, E2 0, E3 0, E4 0} C_DIS
LIN {X 64.118, Y 52.557, Z 58.25, A 0, B 90, C 0, E1 0, E2 0, E3 0, E4 0} C_DIS
LIN {X 66.41, Y 51.368, Z 58.25, A 0, B 90, C 0, E1 0, E2 0, E3 0, E4 0} C_DIS
LIN {X 68.632, Y 50.053, Z 58.25, A 0, B 90, C 0, E1 0, E2 0, E3 0, E4 0} C_DIS
LIN {X 70.756, Y 48.586, Z 58.25, A 0, B 90, C 0, E1 0, E2 0, E3 0, E4 0} C_DIS
LIN {X 72.719, Y 46.911, Z 58.25, A 0, B 90, C 0, E1 0, E2 0, E3 0, E4 0} C_DIS
LIN {X 74.431, Y 44.981, Z 58.25, A 0, B 90, C 0, E1 0, E2 0, E3 0, E4 0} C_DIS
LIN {X 75.881, Y 42.846, Z 58.25, A 0, B 90, C 0, E1 0, E2 0, E3 0, E4 0} C_DIS
LIN {X 77.117, Y 40.58, Z 58.25, A 0, B 90, C 0, E1 0, E2 0, E3 0, E4 0} C_DIS
LIN {X 78.167, Y 38.221, Z 58.25, A 0, B 90, C 0, E1 0, E2 0, E3 0, E4 0} C_DIS
LIN {X 79.044, Y 35.793, Z 58.25, A 0, B 90, C 0, E1 0, E2 0, E3 0, E4 0} C_DIS
LIN {X 79.753, Y 33.311, Z 58.25, A 0, B 90, C 0, E1 0, E2 0, E3 0, E4 0} C_DIS
LIN {X 80.297, Y 30.787, Z 58.25, A 0, B 90, C 0, E1 0, E2 0, E3 0, E4 0} C_DIS
LIN {X 80.681, Y 28.234, Z 58.25, A 0, B 90, C 0, E1 0, E2 0, E3 0, E4 0} C_DIS
LIN {X 80.911, Y 25.662, Z 58.25, A 0, B 90, C 0, E1 0, E2 0, E3 0, E4 0} C_DIS
LIN {X 80.999, Y 23.082, Z 58.25, A 0, B 90, C 0, E1 0, E2 0, E3 0, E4 0} C_DIS
LIN {X 80.961, Y 20.5, Z 58.25, A 0, B 90, C 0, E1 0, E2 0, E3 0, E4 0} C_DIS
LIN {X 80.827, Y 17.921, Z 58.25, A 0, B 90, C 0, E1 0, E2 0, E3 0, E4 0} C_DIS
LIN {X 80.642, Y 15.346, Z 58.25, A 0, B 90, C 0, E1 0, E2 0, E3 0, E4 0} C_DIS
LIN {X 80.439, Y 12.771, Z 58.25, A 0, B 90, C 0, E1 0, E2 0, E3 0, E4 0} C_DIS
LIN {X 80.216, Y 10.199, Z 58.25, A 0, B 90, C 0, E1 0, E2 0, E3 0, E4 0} C_DIS
LIN {X 79.947, Y 7.631, Z 58.25, A 0, B 90, C 0, E1 0, E2 0, E3 0, E4 0} C_DIS
LIN {X 79.611, Y 5.07, Z 58.25, A 0, B 90, C 0, E1 0, E2 0, E3 0, E4 0} C_DIS
LIN {X 79.197, Y 2.522, Z 58.25, A 0, B 90, C 0, E1 0, E2 0, E3 0, E4 0} C_DIS
LIN {X 78.682, Y 0, Z 58.25, A 0, B 90, C 0, E1 0, E2 0, E3 0, E4 0} C_DIS
LIN {X 77.926, Y -2.426, Z 58.25, A 0, B 90, C 0, E1 0, E2 0, E3 0, E4 0} C_DIS
LIN {X 77.221, Y -4.91, Z 58.25, A 0, B 90, C 0, E1 0, E2 0, E3 0, E4 0} C_DIS
LIN {X 76.421, Y -7.365, Z 58.25, A 0, B 90, C 0, E1 0, E2 0, E3 0, E4 0} C_DIS
LIN {X 75.505, Y -9.779, Z 58.25, A 0, B 90, C 0, E1 0, E2 0, E3 0, E4 0} C_DIS
LIN {X 74.423, Y -12.123, Z 58.25, A 0, B 90, C 0, E1 0, E2 0, E3 0, E4 0} C_DIS
LIN {X 73.137, Y -14.361, Z 58.25, A 0, B 90, C 0, E1 0, E2 0, E3 0, E4 0} C_DIS
LIN {X 71.725, Y -16.523, Z 58.25, A 0, B 90, C 0, E1 0, E2 0, E3 0, E4 0} C_DIS
LIN {X 70.284, Y -18.666, Z 58.25, A 0, B 90, C 0, E1 0, E2 0, E3 0, E4 0} C_DIS
LIN {X 68.867, Y -20.824, Z 58.25, A 0, B 90, C 0, E1 0, E2 0, E3 0, E4 0} C_DIS
LIN {X 67.505, Y -23.018, Z 58.25, A 0, B 90, C 0, E1 0, E2 0, E3 0, E4 0} C_DIS
LIN {X 66.22, Y -25.257, Z 58.25, A 0, B 90, C 0, E1 0, E2 0, E3 0, E4 0} C_DIS
LIN {X 65.021, Y -27.544, Z 58.25, A 0, B 90, C 0, E1 0, E2 0, E3 0, E4 0} C_DIS
LIN {X 63.909, Y -29.875, Z 58.25, A 0, B 90, C 0, E1 0, E2 0, E3 0, E4 0} C_DIS
LIN {X 62.876, Y -32.241, Z 58.25, A 0, B 90, C 0, E1 0, E2 0, E3 0, E4 0} C_DIS
LIN {X 61.915, Y -34.638, Z 58.25, A 0, B 90, C 0, E1 0, E2 0, E3 0, E4 0} C_DIS
LIN {X 61.026, Y -37.062, Z 58.25, A 0, B 90, C 0, E1 0, E2 0, E3 0, E4 0} C_DIS
LIN {X 60.218, Y -39.515, Z 58.25, A 0, B 90, C 0, E1 0, E2 0, E3 0, E4 0} C_DIS
LIN {X 59.506, Y -41.997, Z 58.25, A 0, B 90, C 0, E1 0, E2 0, E3 0, E4 0} C_DIS
LIN {X 58.874, Y -44.5, Z 58.25, A 0, B 90, C 0, E1 0, E2 0, E3 0, E4 0} C_DIS
LIN {X 58.277, Y -47.013, Z 58.25, A 0, B 90, C 0, E1 0, E2 0, E3 0, E4 0} C_DIS
LIN {X 57.666, Y -49.522, Z 58.25, A 0, B 90, C 0, E1 0, E2 0, E3 0, E4 0} C_DIS
LIN {X 57.011, Y -52.019, Z 58.25, A 0, B 90, C 0, E1 0, E2 0, E3 0, E4 0} C_DIS
LIN {X 56.292, Y -54.499, Z 58.25, A 0, B 90, C 0, E1 0, E2 0, E3 0, E4 0} C_DIS
LIN {X 55.495, Y -56.955, Z 58.25, A 0, B 90, C 0, E1 0, E2 0, E3 0, E4 0} C_DIS
LIN {X 54.612, Y -59.382, Z 58.25, A 0, B 90, C 0, E1 0, E2 0, E3 0, E4 0} C_DIS
LIN {X 53.635, Y -61.772, Z 58.25, A 0, B 90, C 0, E1 0, E2 0, E3 0, E4 0} C_DIS
LIN {X 52.557, Y -64.118, Z 58.25, A 0, B 90, C 0, E1 0, E2 0, E3 0, E4 0} C_DIS
LIN {X 51.368, Y -66.41, Z 58.25, A 0, B 90, C 0, E1 0, E2 0, E3 0, E4 0} C_DIS
LIN {X 50.053, Y -68.632, Z 58.25, A 0, B 90, C 0, E1 0, E2 0, E3 0, E4 0} C_DIS
LIN {X 48.586, Y -70.756, Z 58.25, A 0, B 90, C 0, E1 0, E2 0, E3 0, E4 0} C_DIS
LIN {X 46.911, Y -72.719, Z 58.25, A 0, B 90, C 0, E1 0, E2 0, E3 0, E4 0} C_DIS
LIN {X 44.981, Y -74.431, Z 58.25, A 0, B 90, C 0, E1 0, E2 0, E3 0, E4 0} C_DIS
LIN {X 42.846, Y -75.881, Z 58.25, A 0, B 90, C 0, E1 0, E2 0, E3 0, E4 0} C_DIS
LIN {X 40.58, Y -77.117, Z 58.25, A 0, B 90, C 0, E1 0, E2 0, E3 0, E4 0} C_DIS
LIN {X 38.221, Y -78.167, Z 58.25, A 0, B 90, C 0, E1 0, E2 0, E3 0, E4 0} C_DIS
LIN {X 35.793, Y -79.044, Z 58.25, A 0, B 90, C 0, E1 0, E2 0, E3 0, E4 0} C_DIS
LIN {X 33.311, Y -79.753, Z 58.25, A 0, B 90, C 0, E1 0, E2 0, E3 0, E4 0} C_DIS
LIN {X 30.787, Y -80.297, Z 58.25, A 0, B 90, C 0, E1 0, E2 0, E3 0, E4 0} C_DIS
LIN {X 28.234, Y -80.681, Z 58.25, A 0, B 90, C 0, E1 0, E2 0, E3 0, E4 0} C_DIS
LIN {X 25.662, Y -80.911, Z 58.25, A 0, B 90, C 0, E1 0, E2 0, E3 0, E4 0} C_DIS
LIN {X 23.082, Y -80.999, Z 58.25, A 0, B 90, C 0, E1 0, E2 0, E3 0, E4 0} C_DIS
LIN {X 20.5, Y -80.961, Z 58.25, A 0, B 90, C 0, E1 0, E2 0, E3 0, E4 0} C_DIS
LIN {X 17.921, Y -80.827, Z 58.25, A 0, B 90, C 0, E1 0, E2 0, E3 0, E4 0} C_DIS
LIN {X 15.346, Y -80.642, Z 58.25, A 0, B 90, C 0, E1 0, E2 0, E3 0, E4 0} C_DIS
LIN {X 12.771, Y -80.439, Z 58.25, A 0, B 90, C 0, E1 0, E2 0, E3 0, E4 0} C_DIS
LIN {X 10.199, Y -80.216, Z 58.25, A 0, B 90, C 0, E1 0, E2 0, E3 0, E4 0} C_DIS
LIN {X 7.631, Y -79.947, Z 58.25, A 0, B 90, C 0, E1 0, E2 0, E3 0, E4 0} C_DIS
LIN {X 5.07, Y -79.611, Z 58.25, A 0, B 90, C 0, E1 0, E2 0, E3 0, E4 0} C_DIS
LIN {X 2.522, Y -79.197, Z 58.25, A 0, B 90, C 0, E1 0, E2 0, E3 0, E4 0} C_DIS
LIN {X 0, Y -78.682, Z 58.25, A 0, B 90, C 0, E1 0, E2 0, E3 0, E4 0} C_DIS
LIN {X -2.426, Y -77.926, Z 58.25, A 0, B 90, C 0, E1 0, E2 0, E3 0, E4 0} C_DIS
LIN {X -4.91, Y -77.221, Z 58.25, A 0, B 90, C 0, E1 0, E2 0, E3 0, E4 0} C_DIS
LIN {X -7.365, Y -76.421, Z 58.25, A 0, B 90, C 0, E1 0, E2 0, E3 0, E4 0} C_DIS
LIN {X -9.779, Y -75.505, Z 58.25, A 0, B 90, C 0, E1 0, E2 0, E3 0, E4 0} C_DIS
LIN {X -12.123, Y -74.423, Z 58.25, A 0, B 90, C 0, E1 0, E2 0, E3 0, E4 0} C_DIS
LIN {X -14.361, Y -73.137, Z 58.25, A 0, B 90, C 0, E1 0, E2 0, E3 0, E4 0} C_DIS
LIN {X -16.523, Y -71.725, Z 58.25, A 0, B 90, C 0, E1 0, E2 0, E3 0, E4 0} C_DIS
LIN {X -18.666, Y -70.284, Z 58.25, A 0, B 90, C 0, E1 0, E2 0, E3 0, E4 0} C_DIS
LIN {X -20.824, Y -68.867, Z 58.25, A 0, B 90, C 0, E1 0, E2 0, E3 0, E4 0} C_DIS
LIN {X -23.018, Y -67.505, Z 58.25, A 0, B 90, C 0, E1 0, E2 0, E3 0, E4 0} C_DIS
LIN {X -25.257, Y -66.22, Z 58.25, A 0, B 90, C 0, E1 0, E2 0, E3 0, E4 0} C_DIS
LIN {X -27.544, Y -65.021, Z 58.25, A 0, B 90, C 0, E1 0, E2 0, E3 0, E4 0} C_DIS
LIN {X -29.875, Y -63.909, Z 58.25, A 0, B 90, C 0, E1 0, E2 0, E3 0, E4 0} C_DIS
LIN {X -32.241, Y -62.876, Z 58.25, A 0, B 90, C 0, E1 0, E2 0, E3 0, E4 0} C_DIS
LIN {X -34.638, Y -61.915, Z 58.25, A 0, B 90, C 0, E1 0, E2 0, E3 0, E4 0} C_DIS
LIN {X -37.062, Y -61.026, Z 58.25, A 0, B 90, C 0, E1 0, E2 0, E3 0, E4 0} C_DIS
LIN {X -39.515, Y -60.218, Z 58.25, A 0, B 90, C 0, E1 0, E2 0, E3 0, E4 0} C_DIS
LIN {X -41.997, Y -59.506, Z 58.25, A 0, B 90, C 0, E1 0, E2 0, E3 0, E4 0} C_DIS
LIN {X -44.5, Y -58.874, Z 58.25, A 0, B 90, C 0, E1 0, E2 0, E3 0, E4 0} C_DIS
LIN {X -47.013, Y -58.277, Z 58.25, A 0, B 90, C 0, E1 0, E2 0, E3 0, E4 0} C_DIS
LIN {X -49.522, Y -57.666, Z 58.25, A 0, B 90, C 0, E1 0, E2 0, E3 0, E4 0} C_DIS
LIN {X -52.019, Y -57.011, Z 58.25, A 0, B 90, C 0, E1 0, E2 0, E3 0, E4 0} C_DIS
LIN {X -54.499, Y -56.292, Z 58.25, A 0, B 90, C 0, E1 0, E2 0, E3 0, E4 0} C_DIS
LIN {X -56.955, Y -55.495, Z 58.25, A 0, B 90, C 0, E1 0, E2 0, E3 0, E4 0} C_DIS
LIN {X -59.382, Y -54.612, Z 58.25, A 0, B 90, C 0, E1 0, E2 0, E3 0, E4 0} C_DIS
LIN {X -61.772, Y -53.635, Z 58.25, A 0, B 90, C 0, E1 0, E2 0, E3 0, E4 0} C_DIS
LIN {X -64.118, Y -52.557, Z 58.25, A 0, B 90, C 0, E1 0, E2 0, E3 0, E4 0} C_DIS
LIN {X -66.41, Y -51.368, Z 58.25, A 0, B 90, C 0, E1 0, E2 0, E3 0, E4 0} C_DIS
LIN {X -68.632, Y -50.053, Z 58.25, A 0, B 90, C 0, E1 0, E2 0, E3 0, E4 0} C_DIS
LIN {X -70.756, Y -48.586, Z 58.25, A 0, B 90, C 0, E1 0, E2 0, E3 0, E4 0} C_DIS
LIN {X -72.719, Y -46.911, Z 58.25, A 0, B 90, C 0, E1 0, E2 0, E3 0, E4 0} C_DIS
LIN {X -74.431, Y -44.981, Z 58.25, A 0, B 90, C 0, E1 0, E2 0, E3 0, E4 0} C_DIS
LIN {X -75.881, Y -42.846, Z 58.25, A 0, B 90, C 0, E1 0, E2 0, E3 0, E4 0} C_DIS
LIN {X -77.117, Y -40.58, Z 58.25, A 0, B 90, C 0, E1 0, E2 0, E3 0, E4 0} C_DIS
LIN {X -78.167, Y -38.221, Z 58.25, A 0, B 90, C 0, E1 0, E2 0, E3 0, E4 0} C_DIS
LIN {X -79.044, Y -35.793, Z 58.25, A 0, B 90, C 0, E1 0, E2 0, E3 0, E4 0} C_DIS
LIN {X -79.753, Y -33.311, Z 58.25, A 0, B 90, C 0, E1 0, E2 0, E3 0, E4 0} C_DIS
LIN {X -80.297, Y -30.787, Z 58.25, A 0, B 90, C 0, E1 0, E2 0, E3 0, E4 0} C_DIS
LIN {X -80.681, Y -28.234, Z 58.25, A 0, B 90, C 0, E1 0, E2 0, E3 0, E4 0} C_DIS
LIN {X -80.911, Y -25.662, Z 58.25, A 0, B 90, C 0, E1 0, E2 0, E3 0, E4 0} C_DIS
LIN {X -80.999, Y -23.082, Z 58.25, A 0, B 90, C 0, E1 0, E2 0, E3 0, E4 0} C_DIS
LIN {X -80.961, Y -20.5, Z 58.25, A 0, B 90, C 0, E1 0, E2 0, E3 0, E4 0} C_DIS
LIN {X -80.827, Y -17.921, Z 58.25, A 0, B 90, C 0, E1 0, E2 0, E3 0, E4 0} C_DIS
LIN {X -80.642, Y -15.346, Z 58.25, A 0, B 90, C 0, E1 0, E2 0, E3 0, E4 0} C_DIS
LIN {X -80.439, Y -12.771, Z 58.25, A 0, B 90, C 0, E1 0, E2 0, E3 0, E4 0} C_DIS
LIN {X -80.216, Y -10.199, Z 58.25, A 0, B 90, C 0, E1 0, E2 0, E3 0, E4 0} C_DIS
LIN {X -79.947, Y -7.631, Z 58.25, A 0, B 90, C 0, E1 0, E2 0, E3 0, E4 0} C_DIS
LIN {X -79.611, Y -5.07, Z 58.25, A 0, B 90, C 0, E1 0, E2 0, E3 0, E4 0} C_DIS
LIN {X -79.197, Y -2.522, Z 58.25, A 0, B 90, C 0, E1 0, E2 0, E3 0, E4 0} C_DIS
LIN {X -78.707, Y 0, Z 60.75, A 0, B 90, C 0, E1 0, E2 0, E3 0, E4 0} C_DIS
LIN {X -77.915, Y 2.418, Z 60.75, A 0, B 90, C 0, E1 0, E2 0, E3 0, E4 0} C_DIS
LIN {X -77.18, Y 4.903, Z 60.75, A 0, B 90, C 0, E1 0, E2 0, E3 0, E4 0} C_DIS
LIN {X -76.349, Y 7.357, Z 60.75, A 0, B 90, C 0, E1 0, E2 0, E3 0, E4 0} C_DIS
LIN {X -75.401, Y 9.768, Z 60.75, A 0, B 90, C 0, E1 0, E2 0, E3 0, E4 0} C_DIS
LIN {X -74.286, Y 12.106, Z 60.75, A 0, B 90, C 0, E1 0, E2 0, E3 0, E4 0} C_DIS
LIN {X -72.965, Y 14.335, Z 60.75, A 0, B 90, C 0, E1 0, E2 0, E3 0, E4 0} C_DIS
LIN {X -71.521, Y 16.486, Z 60.75, A 0, B 90, C 0, E1 0, E2 0, E3 0, E4 0} C_DIS
LIN {X -70.051, Y 18.62, Z 60.75, A 0, B 90, C 0, E1 0, E2 0, E3 0, E4 0} C_DIS
LIN {X -68.608, Y 20.772, Z 60.75, A 0, B 90, C 0, E1 0, E2 0, E3 0, E4 0} C_DIS
LIN {X -67.224, Y 22.962, Z 60.75, A 0, B 90, C 0, E1 0, E2 0, E3 0, E4 0} C_DIS
LIN {X -65.922, Y 25.202, Z 60.75, A 0, B 90, C 0, E1 0, E2 0, E3 0, E4 0} C_DIS
LIN {X -64.712, Y 27.493, Z 60.75, A 0, B 90, C 0, E1 0, E2 0, E3 0, E4 0} C_DIS
LIN {X -63.595, Y 29.831, Z 60.75, A 0, B 90, C 0, E1 0, E2 0, E3 0, E4 0} C_DIS
LIN {X -62.563, Y 32.208, Z 60.75, A 0, B 90, C 0, E1 0, E2 0, E3 0, E4 0} C_DIS
LIN {X -61.61, Y 34.617, Z 60.75, A 0, B 90, C 0, E1 0, E2 0, E3 0, E4 0} C_DIS
LIN {X -60.733, Y 37.056, Z 60.75, A 0, B 90, C 0, E1 0, E2 0, E3 0, E4 0} C_DIS
LIN {X -59.946, Y 39.524, Z 60.75, A 0, B 90, C 0, E1 0, E2 0, E3 0, E4 0} C_DIS
LIN {X -59.26, Y 42.023, Z 60.75, A 0, B 90, C 0, E1 0, E2 0, E3 0, E4 0} C_DIS
LIN {X -58.659, Y 44.543, Z 60.75, A 0, B 90, C 0, E1 0, E2 0, E3 0, E4 0} C_DIS
LIN {X -58.095, Y 47.072, Z 60.75, A 0, B 90, C 0, E1 0, E2 0, E3 0, E4 0} C_DIS
LIN {X -57.519, Y 49.598, Z 60.75, A 0, B 90, C 0, E1 0, E2 0, E3 0, E4 0} C_DIS
LIN {X -56.898, Y 52.114, Z 60.75, A 0, B 90, C 0, E1 0, E2 0, E3 0, E4 0} C_DIS
LIN {X -56.211, Y 54.612, Z 60.75, A 0, B 90, C 0, E1 0, E2 0, E3 0, E4 0} C_DIS
LIN {X -55.447, Y 57.088, Z 60.75, A 0, B 90, C 0, E1 0, E2 0, E3 0, E4 0} C_DIS
LIN {X -54.596, Y 59.535, Z 60.75, A 0, B 90, C 0, E1 0, E2 0, E3 0, E4 0} C_DIS
LIN {X -53.649, Y 61.947, Z 60.75, A 0, B 90, C 0, E1 0, E2 0, E3 0, E4 0} C_DIS
LIN {X -52.599, Y 64.316, Z 60.75, A 0, B 90, C 0, E1 0, E2 0, E3 0, E4 0} C_DIS
LIN {X -51.436, Y 66.631, Z 60.75, A 0, B 90, C 0, E1 0, E2 0, E3 0, E4 0} C_DIS
LIN {X -50.145, Y 68.877, Z 60.75, A 0, B 90, C 0, E1 0, E2 0, E3 0, E4 0} C_DIS
LIN {X -48.698, Y 71.026, Z 60.75, A 0, B 90, C 0, E1 0, E2 0, E3 0, E4 0} C_DIS
LIN {X -47.039, Y 73.014, Z 60.75, A 0, B 90, C 0, E1 0, E2 0, E3 0, E4 0} C_DIS
LIN {X -45.115, Y 74.746, Z 60.75, A 0, B 90, C 0, E1 0, E2 0, E3 0, E4 0} C_DIS
LIN {X -42.978, Y 76.209, Z 60.75, A 0, B 90, C 0, E1 0, E2 0, E3 0, E4 0} C_DIS
LIN {X -40.706, Y 77.452, Z 60.75, A 0, B 90, C 0, E1 0, E2 0, E3 0, E4 0} C_DIS
LIN {X -38.339, Y 78.505, Z 60.75, A 0, B 90, C 0, E1 0, E2 0, E3 0, E4 0} C_DIS
LIN {X -35.9, Y 79.38, Z 60.75, A 0, B 90, C 0, E1 0, E2 0, E3 0, E4 0} C_DIS
LIN {X -33.407, Y 80.082, Z 60.75, A 0, B 90, C 0, E1 0, E2 0, E3 0, E4 0} C_DIS
LIN {X -30.872, Y 80.616, Z 60.75, A 0, B 90, C 0, E1 0, E2 0, E3 0, E4 0} C_DIS
LIN {X -28.307, Y 80.986, Z 60.75, A 0, B 90, C 0, E1 0, E2 0, E3 0, E4 0} C_DIS
LIN {X -25.725, Y 81.199, Z 60.75, A 0, B 90, C 0, E1 0, E2 0, E3 0, E4 0} C_DIS
LIN {X -23.135, Y 81.266, Z 60.75, A 0, B 90, C 0, E1 0, E2 0, E3 0, E4 0} C_DIS
LIN {X -20.545, Y 81.204, Z 60.75, A 0, B 90, C 0, E1 0, E2 0, E3 0, E4 0} C_DIS
LIN {X -17.959, Y 81.045, Z 60.75, A 0, B 90, C 0, E1 0, E2 0, E3 0, E4 0} C_DIS
LIN {X -15.377, Y 80.832, Z 60.75, A 0, B 90, C 0, E1 0, E2 0, E3 0, E4 0} C_DIS
LIN {X -12.796, Y 80.601, Z 60.75, A 0, B 90, C 0, E1 0, E2 0, E3 0, E4 0} C_DIS
LIN {X -10.217, Y 80.352, Z 60.75, A 0, B 90, C 0, E1 0, E2 0, E3 0, E4 0} C_DIS
LIN {X -7.642, Y 80.056, Z 60.75, A 0, B 90, C 0, E1 0, E2 0, E3 0, E4 0} C_DIS
LIN {X -5.077, Y 79.693, Z 60.75, A 0, B 90, C 0, E1 0, E2 0, E3 0, E4 0} C_DIS
LIN {X -2.524, Y 79.252, Z 60.75, A 0, B 90, C 0, E1 0, E2 0, E3 0, E4 0} C_DIS
LIN {X 0, Y 78.707, Z 60.75, A 0, B 90, C 0, E1 0, E2 0, E3 0, E4 0} C_DIS
LIN {X 2.418, Y 77.915, Z 60.75, A 0, B 90, C 0, E1 0, E2 0, E3 0, E4 0} C_DIS
LIN {X 4.903, Y 77.18, Z 60.75, A 0, B 90, C 0, E1 0, E2 0, E3 0, E4 0} C_DIS
LIN {X 7.357, Y 76.349, Z 60.75, A 0, B 90, C 0, E1 0, E2 0, E3 0, E4 0} C_DIS
LIN {X 9.768, Y 75.401, Z 60.75, A 0, B 90, C 0, E1 0, E2 0, E3 0, E4 0} C_DIS
LIN {X 12.106, Y 74.286, Z 60.75, A 0, B 90, C 0, E1 0, E2 0, E3 0, E4 0} C_DIS
LIN {X 14.335, Y 72.965, Z 60.75, A 0, B 90, C 0, E1 0, E2 0, E3 0, E4 0} C_DIS
LIN {X 16.486, Y 71.521, Z 60.75, A 0, B 90, C 0, E1 0, E2 0, E3 0, E4 0} C_DIS
LIN {X 18.62, Y 70.051, Z 60.75, A 0, B 90, C 0, E1 0, E2 0, E3 0, E4 0} C_DIS
LIN {X 20.772, Y 68.608, Z 60.75, A 0, B 90, C 0, E1 0, E2 0, E3 0, E4 0} C_DIS
LIN {X 22.962, Y 67.224, Z 60.75, A 0, B 90, C 0, E1 0, E2 0, E3 0, E4 0} C_DIS
LIN {X 25.202, Y 65.922, Z 60.75, A 0, B 90, C 0, E1 0, E2 0, E3 0, E4 0} C_DIS
LIN {X 27.493, Y 64.712, Z 60.75, A 0, B 90, C 0, E1 0, E2 0, E3 0, E4 0} C_DIS
LIN {X 29.831, Y 63.595, Z 60.75, A 0, B 90, C 0, E1 0, E2 0, E3 0, E4 0} C_DIS
LIN {X 32.208, Y 62.563, Z 60.75, A 0, B 90, C 0, E1 0, E2 0, E3 0, E4 0} C_DIS
LIN {X 34.617, Y 61.61, Z 60.75, A 0, B 90, C 0, E1 0, E2 0, E3 0, E4 0} C_DIS
LIN {X 37.056, Y 60.733, Z 60.75, A 0, B 90, C 0, E1 0, E2 0, E3 0, E4 0} C_DIS
LIN {X 39.524, Y 59.946, Z 60.75, A 0, B 90, C 0, E1 0, E2 0, E3 0, E4 0} C_DIS
LIN {X 42.023, Y 59.26, Z 60.75, A 0, B 90, C 0, E1 0, E2 0, E3 0, E4 0} C_DIS
LIN {X 44.543, Y 58.659, Z 60.75, A 0, B 90, C 0, E1 0, E2 0, E3 0, E4 0} C_DIS
LIN {X 47.072, Y 58.095, Z 60.75, A 0, B 90, C 0, E1 0, E2 0, E3 0, E4 0} C_DIS
LIN {X 49.598, Y 57.519, Z 60.75, A 0, B 90, C 0, E1 0, E2 0, E3 0, E4 0} C_DIS
LIN {X 52.114, Y 56.898, Z 60.75, A 0, B 90, C 0, E1 0, E2 0, E3 0, E4 0} C_DIS
LIN {X 54.612, Y 56.211, Z 60.75, A 0, B 90, C 0, E1 0, E2 0, E3 0, E4 0} C_DIS
LIN {X 57.088, Y 55.447, Z 60.75, A 0, B 90, C 0, E1 0, E2 0, E3 0, E4 0} C_DIS
LIN {X 59.535, Y 54.596, Z 60.75, A 0, B 90, C 0, E1 0, E2 0, E3 0, E4 0} C_DIS
LIN {X 61.947, Y 53.649, Z 60.75, A 0, B 90, C 0, E1 0, E2 0, E3 0, E4 0} C_DIS
LIN {X 64.316, Y 52.599, Z 60.75, A 0, B 90, C 0, E1 0, E2 0, E3 0, E4 0} C_DIS
LIN {X 66.631, Y 51.436, Z 60.75, A 0, B 90, C 0, E1 0, E2 0, E3 0, E4 0} C_DIS
LIN {X 68.877, Y 50.145, Z 60.75, A 0, B 90, C 0, E1 0, E2 0, E3 0, E4 0} C_DIS
LIN {X 71.026, Y 48.698, Z 60.75, A 0, B 90, C 0, E1 0, E2 0, E3 0, E4 0} C_DIS
LIN {X 73.014, Y 47.039, Z 60.75, A 0, B 90, C 0, E1 0, E2 0, E3 0, E4 0} C_DIS
LIN {X 74.746, Y 45.115, Z 60.75, A 0, B 90, C 0, E1 0, E2 0, E3 0, E4 0} C_DIS
LIN {X 76.209, Y 42.978, Z 60.75, A 0, B 90, C 0, E1 0, E2 0, E3 0, E4 0} C_DIS
LIN {X 77.452, Y 40.706, Z 60.75, A 0, B 90, C 0, E1 0, E2 0, E3 0, E4 0} C_DIS
LIN {X 78.505, Y 38.339, Z 60.75, A 0, B 90, C 0, E1 0, E2 0, E3 0, E4 0} C_DIS
LIN {X 79.38, Y 35.9, Z 60.75, A 0, B 90, C 0, E1 0, E2 0, E3 0, E4 0} C_DIS
LIN {X 80.082, Y 33.407, Z 60.75, A 0, B 90, C 0, E1 0, E2 0, E3 0, E4 0} C_DIS
LIN {X 80.616, Y 30.872, Z 60.75, A 0, B 90, C 0, E1 0, E2 0, E3 0, E4 0} C_DIS
LIN {X 80.986, Y 28.307, Z 60.75, A 0, B 90, C 0, E1 0, E2 0, E3 0, E4 0} C_DIS
LIN {X 81.199, Y 25.725, Z 60.75, A 0, B 90, C 0, E1 0, E2 0, E3 0, E4 0} C_DIS
LIN {X 81.266, Y 23.135, Z 60.75, A 0, B 90, C 0, E1 0, E2 0, E3 0, E4 0} C_DIS
LIN {X 81.204, Y 20.545, Z 60.75, A 0, B 90, C 0, E1 0, E2 0, E3 0, E4 0} C_DIS
LIN {X 81.045, Y 17.959, Z 60.75, A 0, B 90, C 0, E1 0, E2 0, E3 0, E4 0} C_DIS
LIN {X 80.832, Y 15.377, Z 60.75, A 0, B 90, C 0, E1 0, E2 0, E3 0, E4 0} C_DIS
LIN {X 80.601, Y 12.796, Z 60.75, A 0, B 90, C 0, E1 0, E2 0, E3 0, E4 0} C_DIS
LIN {X 80.352, Y 10.217, Z 60.75, A 0, B 90, C 0, E1 0, E2 0, E3 0, E4 0} C_DIS
LIN {X 80.056, Y 7.642, Z 60.75, A 0, B 90, C 0, E1 0, E2 0, E3 0, E4 0} C_DIS
LIN {X 79.693, Y 5.077, Z 60.75, A 0, B 90, C 0, E1 0, E2 0, E3 0, E4 0} C_DIS
LIN {X 79.252, Y 2.524, Z 60.75, A 0, B 90, C 0, E1 0, E2 0, E3 0, E4 0} C_DIS
LIN {X 78.707, Y 0, Z 60.75, A 0, B 90, C 0, E1 0, E2 0, E3 0, E4 0} C_DIS
LIN {X 77.915, Y -2.418, Z 60.75, A 0, B 90, C 0, E1 0, E2 0, E3 0, E4 0} C_DIS
LIN {X 77.18, Y -4.903, Z 60.75, A 0, B 90, C 0, E1 0, E2 0, E3 0, E4 0} C_DIS
LIN {X 76.349, Y -7.357, Z 60.75, A 0, B 90, C 0, E1 0, E2 0, E3 0, E4 0} C_DIS
LIN {X 75.401, Y -9.768, Z 60.75, A 0, B 90, C 0, E1 0, E2 0, E3 0, E4 0} C_DIS
LIN {X 74.286, Y -12.106, Z 60.75, A 0, B 90, C 0, E1 0, E2 0, E3 0, E4 0} C_DIS
LIN {X 72.965, Y -14.335, Z 60.75, A 0, B 90, C 0, E1 0, E2 0, E3 0, E4 0} C_DIS
LIN {X 71.521, Y -16.486, Z 60.75, A 0, B 90, C 0, E1 0, E2 0, E3 0, E4 0} C_DIS
LIN {X 70.051, Y -18.62, Z 60.75, A 0, B 90, C 0, E1 0, E2 0, E3 0, E4 0} C_DIS
LIN {X 68.608, Y -20.772, Z 60.75, A 0, B 90, C 0, E1 0, E2 0, E3 0, E4 0} C_DIS
LIN {X 67.224, Y -22.962, Z 60.75, A 0, B 90, C 0, E1 0, E2 0, E3 0, E4 0} C_DIS
LIN {X 65.922, Y -25.202, Z 60.75, A 0, B 90, C 0, E1 0, E2 0, E3 0, E4 0} C_DIS
LIN {X 64.712, Y -27.493, Z 60.75, A 0, B 90, C 0, E1 0, E2 0, E3 0, E4 0} C_DIS
LIN {X 63.595, Y -29.831, Z 60.75, A 0, B 90, C 0, E1 0, E2 0, E3 0, E4 0} C_DIS
LIN {X 62.563, Y -32.208, Z 60.75, A 0, B 90, C 0, E1 0, E2 0, E3 0, E4 0} C_DIS
LIN {X 61.61, Y -34.617, Z 60.75, A 0, B 90, C 0, E1 0, E2 0, E3 0, E4 0} C_DIS
LIN {X 60.733, Y -37.056, Z 60.75, A 0, B 90, C 0, E1 0, E2 0, E3 0, E4 0} C_DIS
LIN {X 59.946, Y -39.524, Z 60.75, A 0, B 90, C 0, E1 0, E2 0, E3 0, E4 0} C_DIS
LIN {X 59.26, Y -42.023, Z 60.75, A 0, B 90, C 0, E1 0, E2 0, E3 0, E4 0} C_DIS
LIN {X 58.659, Y -44.543, Z 60.75, A 0, B 90, C 0, E1 0, E2 0, E3 0, E4 0} C_DIS
LIN {X 58.095, Y -47.072, Z 60.75, A 0, B 90, C 0, E1 0, E2 0, E3 0, E4 0} C_DIS
LIN {X 57.519, Y -49.598, Z 60.75, A 0, B 90, C 0, E1 0, E2 0, E3 0, E4 0} C_DIS
LIN {X 56.898, Y -52.114, Z 60.75, A 0, B 90, C 0, E1 0, E2 0, E3 0, E4 0} C_DIS
LIN {X 56.211, Y -54.612, Z 60.75, A 0, B 90, C 0, E1 0, E2 0, E3 0, E4 0} C_DIS
LIN {X 55.447, Y -57.088, Z 60.75, A 0, B 90, C 0, E1 0, E2 0, E3 0, E4 0} C_DIS
LIN {X 54.596, Y -59.535, Z 60.75, A 0, B 90, C 0, E1 0, E2 0, E3 0, E4 0} C_DIS
LIN {X 53.649, Y -61.947, Z 60.75, A 0, B 90, C 0, E1 0, E2 0, E3 0, E4 0} C_DIS
LIN {X 52.599, Y -64.316, Z 60.75, A 0, B 90, C 0, E1 0, E2 0, E3 0, E4 0} C_DIS
LIN {X 51.436, Y -66.631, Z 60.75, A 0, B 90, C 0, E1 0, E2 0, E3 0, E4 0} C_DIS
LIN {X 50.145, Y -68.877, Z 60.75, A 0, B 90, C 0, E1 0, E2 0, E3 0, E4 0} C_DIS
LIN {X 48.698, Y -71.026, Z 60.75, A 0, B 90, C 0, E1 0, E2 0, E3 0, E4 0} C_DIS
LIN {X 47.039, Y -73.014, Z 60.75, A 0, B 90, C 0, E1 0, E2 0, E3 0, E4 0} C_DIS
LIN {X 45.115, Y -74.746, Z 60.75, A 0, B 90, C 0, E1 0, E2 0, E3 0, E4 0} C_DIS
LIN {X 42.978, Y -76.209, Z 60.75, A 0, B 90, C 0, E1 0, E2 0, E3 0, E4 0} C_DIS
LIN {X 40.706, Y -77.452, Z 60.75, A 0, B 90, C 0, E1 0, E2 0, E3 0, E4 0} C_DIS
LIN {X 38.339, Y -78.505, Z 60.75, A 0, B 90, C 0, E1 0, E2 0, E3 0, E4 0} C_DIS
LIN {X 35.9, Y -79.38, Z 60.75, A 0, B 90, C 0, E1 0, E2 0, E3 0, E4 0} C_DIS
LIN {X 33.407, Y -80.082, Z 60.75, A 0, B 90, C 0, E1 0, E2 0, E3 0, E4 0} C_DIS
LIN {X 30.872, Y -80.616, Z 60.75, A 0, B 90, C 0, E1 0, E2 0, E3 0, E4 0} C_DIS
LIN {X 28.307, Y -80.986, Z 60.75, A 0, B 90, C 0, E1 0, E2 0, E3 0, E4 0} C_DIS
LIN {X 25.725, Y -81.199, Z 60.75, A 0, B 90, C 0, E1 0, E2 0, E3 0, E4 0} C_DIS
LIN {X 23.135, Y -81.266, Z 60.75, A 0, B 90, C 0, E1 0, E2 0, E3 0, E4 0} C_DIS
LIN {X 20.545, Y -81.204, Z 60.75, A 0, B 90, C 0, E1 0, E2 0, E3 0, E4 0} C_DIS
LIN {X 17.959, Y -81.045, Z 60.75, A 0, B 90, C 0, E1 0, E2 0, E3 0, E4 0} C_DIS
LIN {X 15.377, Y -80.832, Z 60.75, A 0, B 90, C 0, E1 0, E2 0, E3 0, E4 0} C_DIS
LIN {X 12.796, Y -80.601, Z 60.75, A 0, B 90, C 0, E1 0, E2 0, E3 0, E4 0} C_DIS
LIN {X 10.217, Y -80.352, Z 60.75, A 0, B 90, C 0, E1 0, E2 0, E3 0, E4 0} C_DIS
LIN {X 7.642, Y -80.056, Z 60.75, A 0, B 90, C 0, E1 0, E2 0, E3 0, E4 0} C_DIS
LIN {X 5.077, Y -79.693, Z 60.75, A 0, B 90, C 0, E1 0, E2 0, E3 0, E4 0} C_DIS
LIN {X 2.524, Y -79.252, Z 60.75, A 0, B 90, C 0, E1 0, E2 0, E3 0, E4 0} C_DIS
LIN {X 0, Y -78.707, Z 60.75, A 0, B 90, C 0, E1 0, E2 0, E3 0, E4 0} C_DIS
LIN {X -2.418, Y -77.915, Z 60.75, A 0, B 90, C 0, E1 0, E2 0, E3 0, E4 0} C_DIS
LIN {X -4.903, Y -77.18, Z 60.75, A 0, B 90, C 0, E1 0, E2 0, E3 0, E4 0} C_DIS
LIN {X -7.357, Y -76.349, Z 60.75, A 0, B 90, C 0, E1 0, E2 0, E3 0, E4 0} C_DIS
LIN {X -9.768, Y -75.401, Z 60.75, A 0, B 90, C 0, E1 0, E2 0, E3 0, E4 0} C_DIS
LIN {X -12.106, Y -74.286, Z 60.75, A 0, B 90, C 0, E1 0, E2 0, E3 0, E4 0} C_DIS
LIN {X -14.335, Y -72.965, Z 60.75, A 0, B 90, C 0, E1 0, E2 0, E3 0, E4 0} C_DIS
LIN {X -16.486, Y -71.521, Z 60.75, A 0, B 90, C 0, E1 0, E2 0, E3 0, E4 0} C_DIS
LIN {X -18.62, Y -70.051, Z 60.75, A 0, B 90, C 0, E1 0, E2 0, E3 0, E4 0} C_DIS
LIN {X -20.772, Y -68.608, Z 60.75, A 0, B 90, C 0, E1 0, E2 0, E3 0, E4 0} C_DIS
LIN {X -22.962, Y -67.224, Z 60.75, A 0, B 90, C 0, E1 0, E2 0, E3 0, E4 0} C_DIS
LIN {X -25.202, Y -65.922, Z 60.75, A 0, B 90, C 0, E1 0, E2 0, E3 0, E4 0} C_DIS
LIN {X -27.493, Y -64.712, Z 60.75, A 0, B 90, C 0, E1 0, E2 0, E3 0, E4 0} C_DIS
LIN {X -29.831, Y -63.595, Z 60.75, A 0, B 90, C 0, E1 0, E2 0, E3 0, E4 0} C_DIS
LIN {X -32.208, Y -62.563, Z 60.75, A 0, B 90, C 0, E1 0, E2 0, E3 0, E4 0} C_DIS
LIN {X -34.617, Y -61.61, Z 60.75, A 0, B 90, C 0, E1 0, E2 0, E3 0, E4 0} C_DIS
LIN {X -37.056, Y -60.733, Z 60.75, A 0, B 90, C 0, E1 0, E2 0, E3 0, E4 0} C_DIS
LIN {X -39.524, Y -59.946, Z 60.75, A 0, B 90, C 0, E1 0, E2 0, E3 0, E4 0} C_DIS
LIN {X -42.023, Y -59.26, Z 60.75, A 0, B 90, C 0, E1 0, E2 0, E3 0, E4 0} C_DIS
LIN {X -44.543, Y -58.659, Z 60.75, A 0, B 90, C 0, E1 0, E2 0, E3 0, E4 0} C_DIS
LIN {X -47.072, Y -58.095, Z 60.75, A 0, B 90, C 0, E1 0, E2 0, E3 0, E4 0} C_DIS
LIN {X -49.598, Y -57.519, Z 60.75, A 0, B 90, C 0, E1 0, E2 0, E3 0, E4 0} C_DIS
LIN {X -52.114, Y -56.898, Z 60.75, A 0, B 90, C 0, E1 0, E2 0, E3 0, E4 0} C_DIS
LIN {X -54.612, Y -56.211, Z 60.75, A 0, B 90, C 0, E1 0, E2 0, E3 0, E4 0} C_DIS
LIN {X -57.088, Y -55.447, Z 60.75, A 0, B 90, C 0, E1 0, E2 0, E3 0, E4 0} C_DIS
LIN {X -59.535, Y -54.596, Z 60.75, A 0, B 90, C 0, E1 0, E2 0, E3 0, E4 0} C_DIS
LIN {X -61.947, Y -53.649, Z 60.75, A 0, B 90, C 0, E1 0, E2 0, E3 0, E4 0} C_DIS
LIN {X -64.316, Y -52.599, Z 60.75, A 0, B 90, C 0, E1 0, E2 0, E3 0, E4 0} C_DIS
LIN {X -66.631, Y -51.436, Z 60.75, A 0, B 90, C 0, E1 0, E2 0, E3 0, E4 0} C_DIS
LIN {X -68.877, Y -50.145, Z 60.75, A 0, B 90, C 0, E1 0, E2 0, E3 0, E4 0} C_DIS
LIN {X -71.026, Y -48.698, Z 60.75, A 0, B 90, C 0, E1 0, E2 0, E3 0, E4 0} C_DIS
LIN {X -73.014, Y -47.039, Z 60.75, A 0, B 90, C 0, E1 0, E2 0, E3 0, E4 0} C_DIS
LIN {X -74.746, Y -45.115, Z 60.75, A 0, B 90, C 0, E1 0, E2 0, E3 0, E4 0} C_DIS
LIN {X -76.209, Y -42.978, Z 60.75, A 0, B 90, C 0, E1 0, E2 0, E3 0, E4 0} C_DIS
LIN {X -77.452, Y -40.706, Z 60.75, A 0, B 90, C 0, E1 0, E2 0, E3 0, E4 0} C_DIS
LIN {X -78.505, Y -38.339, Z 60.75, A 0, B 90, C 0, E1 0, E2 0, E3 0, E4 0} C_DIS
LIN {X -79.38, Y -35.9, Z 60.75, A 0, B 90, C 0, E1 0, E2 0, E3 0, E4 0} C_DIS
LIN {X -80.082, Y -33.407, Z 60.75, A 0, B 90, C 0, E1 0, E2 0, E3 0, E4 0} C_DIS
LIN {X -80.616, Y -30.872, Z 60.75, A 0, B 90, C 0, E1 0, E2 0, E3 0, E4 0} C_DIS
LIN {X -80.986, Y -28.307, Z 60.75, A 0, B 90, C 0, E1 0, E2 0, E3 0, E4 0} C_DIS
LIN {X -81.199, Y -25.725, Z 60.75, A 0, B 90, C 0, E1 0, E2 0, E3 0, E4 0} C_DIS
LIN {X -81.266, Y -23.135, Z 60.75, A 0, B 90, C 0, E1 0, E2 0, E3 0, E4 0} C_DIS
LIN {X -81.204, Y -20.545, Z 60.75, A 0, B 90, C 0, E1 0, E2 0, E3 0, E4 0} C_DIS
LIN {X -81.045, Y -17.959, Z 60.75, A 0, B 90, C 0, E1 0, E2 0, E3 0, E4 0} C_DIS
LIN {X -80.832, Y -15.377, Z 60.75, A 0, B 90, C 0, E1 0, E2 0, E3 0, E4 0} C_DIS
LIN {X -80.601, Y -12.796, Z 60.75, A 0, B 90, C 0, E1 0, E2 0, E3 0, E4 0} C_DIS
LIN {X -80.352, Y -10.217, Z 60.75, A 0, B 90, C 0, E1 0, E2 0, E3 0, E4 0} C_DIS
LIN {X -80.056, Y -7.642, Z 60.75, A 0, B 90, C 0, E1 0, E2 0, E3 0, E4 0} C_DIS
LIN {X -79.693, Y -5.077, Z 60.75, A 0, B 90, C 0, E1 0, E2 0, E3 0, E4 0} C_DIS
LIN {X -79.252, Y -2.524, Z 60.75, A 0, B 90, C 0, E1 0, E2 0, E3 0, E4 0} C_DIS
LIN {X -78.741, Y 0, Z 63.25, A 0, B 90, C 0, E1 0, E2 0, E3 0, E4 0} C_DIS
LIN {X -77.914, Y 2.41, Z 63.25, A 0, B 90, C 0, E1 0, E2 0, E3 0, E4 0} C_DIS
LIN {X -77.148, Y 4.895, Z 63.25, A 0, B 90, C 0, E1 0, E2 0, E3 0, E4 0} C_DIS
LIN {X -76.286, Y 7.348, Z 63.25, A 0, B 90, C 0, E1 0, E2 0, E3 0, E4 0} C_DIS
LIN {X -75.306, Y 9.757, Z 63.25, A 0, B 90, C 0, E1 0, E2 0, E3 0, E4 0} C_DIS
LIN {X -74.159, Y 12.089, Z 63.25, A 0, B 90, C 0, E1 0, E2 0, E3 0, E4 0} C_DIS
LIN {X -72.805, Y 14.309, Z 63.25, A 0, B 90, C 0, E1 0, E2 0, E3 0, E4 0} C_DIS
LIN {X -71.33, Y 16.45, Z 63.25, A 0, B 90, C 0, E1 0, E2 0, E3 0, E4 0} C_DIS
LIN {X -69.832, Y 18.575, Z 63.25, A 0, B 90, C 0, E1 0, E2 0, E3 0, E4 0} C_DIS
LIN {X -68.364, Y 20.722, Z 63.25, A 0, B 90, C 0, E1 0, E2 0, E3 0, E4 0} C_DIS
LIN {X -66.959, Y 22.91, Z 63.25, A 0, B 90, C 0, E1 0, E2 0, E3 0, E4 0} C_DIS
LIN {X -65.64, Y 25.151, Z 63.25, A 0, B 90, C 0, E1 0, E2 0, E3 0, E4 0} C_DIS
LIN {X -64.42, Y 27.447, Z 63.25, A 0, B 90, C 0, E1 0, E2 0, E3 0, E4 0} C_DIS
LIN {X -63.298, Y 29.792, Z 63.25, A 0, B 90, C 0, E1 0, E2 0, E3 0, E4 0} C_DIS
LIN {X -62.268, Y 32.18, Z 63.25, A 0, B 90, C 0, E1 0, E2 0, E3 0, E4 0} C_DIS
LIN {X -61.322, Y 34.602, Z 63.25, A 0, B 90, C 0, E1 0, E2 0, E3 0, E4 0} C_DIS
LIN {X -60.459, Y 37.055, Z 63.25, A 0, B 90, C 0, E1 0, E2 0, E3 0, E4 0} C_DIS
LIN {X -59.691, Y 39.539, Z 63.25, A 0, B 90, C 0, E1 0, E2 0, E3 0, E4 0} C_DIS
LIN {X -59.031, Y 42.054, Z 63.25, A 0, B 90, C 0, E1 0, E2 0, E3 0, E4 0} C_DIS
LIN {X -58.46, Y 44.591, Z 63.25, A 0, B 90, C 0, E1 0, E2 0, E3 0, E4 0} C_DIS
LIN {X -57.929, Y 47.136, Z 63.25, A 0, B 90, C 0, E1 0, E2 0, E3 0, E4 0} C_DIS
LIN {X -57.385, Y 49.679, Z 63.25, A 0, B 90, C 0, E1 0, E2 0, E3 0, E4 0} C_DIS
LIN {X -56.796, Y 52.212, Z 63.25, A 0, B 90, C 0, E1 0, E2 0, E3 0, E4 0} C_DIS
LIN {X -56.142, Y 54.729, Z 63.25, A 0, B 90, C 0, E1 0, E2 0, E3 0, E4 0} C_DIS
LIN {X -55.408, Y 57.223, Z 63.25, A 0, B 90, C 0, E1 0, E2 0, E3 0, E4 0} C_DIS
LIN {X -54.587, Y 59.69, Z 63.25, A 0, B 90, C 0, E1 0, E2 0, E3 0, E4 0} C_DIS
LIN {X -53.668, Y 62.123, Z 63.25, A 0, B 90, C 0, E1 0, E2 0, E3 0, E4 0} C_DIS
LIN {X -52.645, Y 64.513, Z 63.25, A 0, B 90, C 0, E1 0, E2 0, E3 0, E4 0} C_DIS
LIN {X -51.507, Y 66.851, Z 63.25, A 0, B 90, C 0, E1 0, E2 0, E3 0, E4 0} C_DIS
LIN {X -50.239, Y 69.121, Z 63.25, A 0, B 90, C 0, E1 0, E2 0, E3 0, E4 0} C_DIS
LIN {X -48.812, Y 71.294, Z 63.25, A 0, B 90, C 0, E1 0, E2 0, E3 0, E4 0} C_DIS
LIN {X -47.167, Y 73.305, Z 63.25, A 0, B 90, C 0, E1 0, E2 0, E3 0, E4 0} C_DIS
LIN {X -45.249, Y 75.058, Z 63.25, A 0, B 90, C 0, E1 0, E2 0, E3 0, E4 0} C_DIS
LIN {X -43.111, Y 76.535, Z 63.25, A 0, B 90, C 0, E1 0, E2 0, E3 0, E4 0} C_DIS
LIN {X -40.832, Y 77.786, Z 63.25, A 0, B 90, C 0, E1 0, E2 0, E3 0, E4 0} C_DIS
LIN {X -38.457, Y 78.842, Z 63.25, A 0, B 90, C 0, E1 0, E2 0, E3 0, E4 0} C_DIS
LIN {X -36.008, Y 79.715, Z 63.25, A 0, B 90, C 0, E1 0, E2 0, E3 0, E4 0} C_DIS
LIN {X -33.503, Y 80.413, Z 63.25, A 0, B 90, C 0, E1 0, E2 0, E3 0, E4 0} C_DIS
LIN {X -30.957, Y 80.938, Z 63.25, A 0, B 90, C 0, E1 0, E2 0, E3 0, E4 0} C_DIS
LIN {X -28.382, Y 81.295, Z 63.25, A 0, B 90, C 0, E1 0, E2 0, E3 0, E4 0} C_DIS
LIN {X -25.789, Y 81.491, Z 63.25, A 0, B 90, C 0, E1 0, E2 0, E3 0, E4 0} C_DIS
LIN {X -23.19, Y 81.538, Z 63.25, A 0, B 90, C 0, E1 0, E2 0, E3 0, E4 0} C_DIS
LIN {X -20.591, Y 81.454, Z 63.25, A 0, B 90, C 0, E1 0, E2 0, E3 0, E4 0} C_DIS
LIN {X -17.997, Y 81.27, Z 63.25, A 0, B 90, C 0, E1 0, E2 0, E3 0, E4 0} C_DIS
LIN {X -15.408, Y 81.03, Z 63.25, A 0, B 90, C 0, E1 0, E2 0, E3 0, E4 0} C_DIS
LIN {X -12.82, Y 80.773, Z 63.25, A 0, B 90, C 0, E1 0, E2 0, E3 0, E4 0} C_DIS
LIN {X -10.234, Y 80.496, Z 63.25, A 0, B 90, C 0, E1 0, E2 0, E3 0, E4 0} C_DIS
LIN {X -7.654, Y 80.174, Z 63.25, A 0, B 90, C 0, E1 0, E2 0, E3 0, E4 0} C_DIS
LIN {X -5.083, Y 79.784, Z 63.25, A 0, B 90, C 0, E1 0, E2 0, E3 0, E4 0} C_DIS
LIN {X -2.526, Y 79.315, Z 63.25, A 0, B 90, C 0, E1 0, E2 0, E3 0, E4 0} C_DIS
LIN {X 0, Y 78.741, Z 63.25, A 0, B 90, C 0, E1 0, E2 0, E3 0, E4 0} C_DIS
LIN {X 2.41, Y 77.914, Z 63.25, A 0, B 90, C 0, E1 0, E2 0, E3 0, E4 0} C_DIS
LIN {X 4.895, Y 77.148, Z 63.25, A 0, B 90, C 0, E1 0, E2 0, E3 0, E4 0} C_DIS
LIN {X 7.348, Y 76.286, Z 63.25, A 0, B 90, C 0, E1 0, E2 0, E3 0, E4 0} C_DIS
LIN {X 9.757, Y 75.306, Z 63.25, A 0, B 90, C 0, E1 0, E2 0, E3 0, E4 0} C_DIS
LIN {X 12.089, Y 74.159, Z 63.25, A 0, B 90, C 0, E1 0, E2 0, E3 0, E4 0} C_DIS
LIN {X 14.309, Y 72.805, Z 63.25, A 0, B 90, C 0, E1 0, E2 0, E3 0, E4 0} C_DIS
LIN {X 16.45, Y 71.33, Z 63.25, A 0, B 90, C 0, E1 0, E2 0, E3 0, E4 0} C_DIS
LIN {X 18.575, Y 69.832, Z 63.25, A 0, B 90, C 0, E1 0, E2 0, E3 0, E4 0} C_DIS
LIN {X 20.722, Y 68.364, Z 63.25, A 0, B 90, C 0, E1 0, E2 0, E3 0, E4 0} C_DIS
LIN {X 22.91, Y 66.959, Z 63.25, A 0, B 90, C 0, E1 0, E2 0, E3 0, E4 0} C_DIS
LIN {X 25.151, Y 65.64, Z 63.25, A 0, B 90, C 0, E1 0, E2 0, E3 0, E4 0} C_DIS
LIN {X 27.447, Y 64.42, Z 63.25, A 0, B 90, C 0, E1 0, E2 0, E3 0, E4 0} C_DIS
LIN {X 29.792, Y 63.298, Z 63.25, A 0, B 90, C 0, E1 0, E2 0, E3 0, E4 0} C_DIS
LIN {X 32.18, Y 62.268, Z 63.25, A 0, B 90, C 0, E1 0, E2 0, E3 0, E4 0} C_DIS
LIN {X 34.602, Y 61.322, Z 63.25, A 0, B 90, C 0, E1 0, E2 0, E3 0, E4 0} C_DIS
LIN {X 37.055, Y 60.459, Z 63.25, A 0, B 90, C 0, E1 0, E2 0, E3 0, E4 0} C_DIS
LIN {X 39.539, Y 59.691, Z 63.25, A 0, B 90, C 0, E1 0, E2 0, E3 0, E4 0} C_DIS
LIN {X 42.054, Y 59.031, Z 63.25, A 0, B 90, C 0, E1 0, E2 0, E3 0, E4 0} C_DIS
LIN {X 44.591, Y 58.46, Z 63.25, A 0, B 90, C 0, E1 0, E2 0, E3 0, E4 0} C_DIS
LIN {X 47.136, Y 57.929, Z 63.25, A 0, B 90, C 0, E1 0, E2 0, E3 0, E4 0} C_DIS
LIN {X 49.679, Y 57.385, Z 63.25, A 0, B 90, C 0, E1 0, E2 0, E3 0, E4 0} C_DIS
LIN {X 52.212, Y 56.796, Z 63.25, A 0, B 90, C 0, E1 0, E2 0, E3 0, E4 0} C_DIS
LIN {X 54.729, Y 56.142, Z 63.25, A 0, B 90, C 0, E1 0, E2 0, E3 0, E4 0} C_DIS
LIN {X 57.223, Y 55.408, Z 63.25, A 0, B 90, C 0, E1 0, E2 0, E3 0, E4 0} C_DIS
LIN {X 59.69, Y 54.587, Z 63.25, A 0, B 90, C 0, E1 0, E2 0, E3 0, E4 0} C_DIS
LIN {X 62.123, Y 53.668, Z 63.25, A 0, B 90, C 0, E1 0, E2 0, E3 0, E4 0} C_DIS
LIN {X 64.513, Y 52.645, Z 63.25, A 0, B 90, C 0, E1 0, E2 0, E3 0, E4 0} C_DIS
LIN {X 66.851, Y 51.507, Z 63.25, A 0, B 90, C 0, E1 0, E2 0, E3 0, E4 0} C_DIS
LIN {X 69.121, Y 50.239, Z 63.25, A 0, B 90, C 0, E1 0, E2 0, E3 0, E4 0} C_DIS
LIN {X 71.294, Y 48.812, Z 63.25, A 0, B 90, C 0, E1 0, E2 0, E3 0, E4 0} C_DIS
LIN {X 73.305, Y 47.167, Z 63.25, A 0, B 90, C 0, E1 0, E2 0, E3 0, E4 0} C_DIS
LIN {X 75.058, Y 45.249, Z 63.25, A 0, B 90, C 0, E1 0, E2 0, E3 0, E4 0} C_DIS
LIN {X 76.535, Y 43.111, Z 63.25, A 0, B 90, C 0, E1 0, E2 0, E3 0, E4 0} C_DIS
LIN {X 77.786, Y 40.832, Z 63.25, A 0, B 90, C 0, E1 0, E2 0, E3 0, E4 0} C_DIS
LIN {X 78.842, Y 38.457, Z 63.25, A 0, B 90, C 0, E1 0, E2 0, E3 0, E4 0} C_DIS
LIN {X 79.715, Y 36.008, Z 63.25, A 0, B 90, C 0, E1 0, E2 0, E3 0, E4 0} C_DIS
LIN {X 80.413, Y 33.503, Z 63.25, A 0, B 90, C 0, E1 0, E2 0, E3 0, E4 0} C_DIS
LIN {X 80.938, Y 30.957, Z 63.25, A 0, B 90, C 0, E1 0, E2 0, E3 0, E4 0} C_DIS
LIN {X 81.295, Y 28.382, Z 63.25, A 0, B 90, C 0, E1 0, E2 0, E3 0, E4 0} C_DIS
LIN {X 81.491, Y 25.789, Z 63.25, A 0, B 90, C 0, E1 0, E2 0, E3 0, E4 0} C_DIS
LIN {X 81.538, Y 23.19, Z 63.25, A 0, B 90, C 0, E1 0, E2 0, E3 0, E4 0} C_DIS
LIN {X 81.454, Y 20.591, Z 63.25, A 0, B 90, C 0, E1 0, E2 0, E3 0, E4 0} C_DIS
LIN {X 81.27, Y 17.997, Z 63.25, A 0, B 90, C 0, E1 0, E2 0, E3 0, E4 0} C_DIS
LIN {X 81.03, Y 15.408, Z 63.25, A 0, B 90, C 0, E1 0, E2 0, E3 0, E4 0} C_DIS
LIN {X 80.773, Y 12.82, Z 63.25, A 0, B 90, C 0, E1 0, E2 0, E3 0, E4 0} C_DIS
LIN {X 80.496, Y 10.234, Z 63.25, A 0, B 90, C 0, E1 0, E2 0, E3 0, E4 0} C_DIS
LIN {X 80.174, Y 7.654, Z 63.25, A 0, B 90, C 0, E1 0, E2 0, E3 0, E4 0} C_DIS
LIN {X 79.784, Y 5.083, Z 63.25, A 0, B 90, C 0, E1 0, E2 0, E3 0, E4 0} C_DIS
LIN {X 79.315, Y 2.526, Z 63.25, A 0, B 90, C 0, E1 0, E2 0, E3 0, E4 0} C_DIS
LIN {X 78.741, Y 0, Z 63.25, A 0, B 90, C 0, E1 0, E2 0, E3 0, E4 0} C_DIS
LIN {X 77.914, Y -2.41, Z 63.25, A 0, B 90, C 0, E1 0, E2 0, E3 0, E4 0} C_DIS
LIN {X 77.148, Y -4.895, Z 63.25, A 0, B 90, C 0, E1 0, E2 0, E3 0, E4 0} C_DIS
LIN {X 76.286, Y -7.348, Z 63.25, A 0, B 90, C 0, E1 0, E2 0, E3 0, E4 0} C_DIS
LIN {X 75.306, Y -9.757, Z 63.25, A 0, B 90, C 0, E1 0, E2 0, E3 0, E4 0} C_DIS
LIN {X 74.159, Y -12.089, Z 63.25, A 0, B 90, C 0, E1 0, E2 0, E3 0, E4 0} C_DIS
LIN {X 72.805, Y -14.309, Z 63.25, A 0, B 90, C 0, E1 0, E2 0, E3 0, E4 0} C_DIS
LIN {X 71.33, Y -16.45, Z 63.25, A 0, B 90, C 0, E1 0, E2 0, E3 0, E4 0} C_DIS
LIN {X 69.832, Y -18.575, Z 63.25, A 0, B 90, C 0, E1 0, E2 0, E3 0, E4 0} C_DIS
LIN {X 68.364, Y -20.722, Z 63.25, A 0, B 90, C 0, E1 0, E2 0, E3 0, E4 0} C_DIS
LIN {X 66.959, Y -22.91, Z 63.25, A 0, B 90, C 0, E1 0, E2 0, E3 0, E4 0} C_DIS
LIN {X 65.64, Y -25.151, Z 63.25, A 0, B 90, C 0, E1 0, E2 0, E3 0, E4 0} C_DIS
LIN {X 64.42, Y -27.447, Z 63.25, A 0, B 90, C 0, E1 0, E2 0, E3 0, E4 0} C_DIS
LIN {X 63.298, Y -29.792, Z 63.25, A 0, B 90, C 0, E1 0, E2 0, E3 0, E4 0} C_DIS
LIN {X 62.268, Y -32.18, Z 63.25, A 0, B 90, C 0, E1 0, E2 0, E3 0, E4 0} C_DIS
LIN {X 61.322, Y -34.602, Z 63.25, A 0, B 90, C 0, E1 0, E2 0, E3 0, E4 0} C_DIS
LIN {X 60.459, Y -37.055, Z 63.25, A 0, B 90, C 0, E1 0, E2 0, E3 0, E4 0} C_DIS
LIN {X 59.691, Y -39.539, Z 63.25, A 0, B 90, C 0, E1 0, E2 0, E3 0, E4 0} C_DIS
LIN {X 59.031, Y -42.054, Z 63.25, A 0, B 90, C 0, E1 0, E2 0, E3 0, E4 0} C_DIS
LIN {X 58.46, Y -44.591, Z 63.25, A 0, B 90, C 0, E1 0, E2 0, E3 0, E4 0} C_DIS
LIN {X 57.929, Y -47.136, Z 63.25, A 0, B 90, C 0, E1 0, E2 0, E3 0, E4 0} C_DIS
LIN {X 57.385, Y -49.679, Z 63.25, A 0, B 90, C 0, E1 0, E2 0, E3 0, E4 0} C_DIS
LIN {X 56.796, Y -52.212, Z 63.25, A 0, B 90, C 0, E1 0, E2 0, E3 0, E4 0} C_DIS
LIN {X 56.142, Y -54.729, Z 63.25, A 0, B 90, C 0, E1 0, E2 0, E3 0, E4 0} C_DIS
LIN {X 55.408, Y -57.223, Z 63.25, A 0, B 90, C 0, E1 0, E2 0, E3 0, E4 0} C_DIS
LIN {X 54.587, Y -59.69, Z 63.25, A 0, B 90, C 0, E1 0, E2 0, E3 0, E4 0} C_DIS
LIN {X 53.668, Y -62.123, Z 63.25, A 0, B 90, C 0, E1 0, E2 0, E3 0, E4 0} C_DIS
LIN {X 52.645, Y -64.513, Z 63.25, A 0, B 90, C 0, E1 0, E2 0, E3 0, E4 0} C_DIS
LIN {X 51.507, Y -66.851, Z 63.25, A 0, B 90, C 0, E1 0, E2 0, E3 0, E4 0} C_DIS
LIN {X 50.239, Y -69.121, Z 63.25, A 0, B 90, C 0, E1 0, E2 0, E3 0, E4 0} C_DIS
LIN {X 48.812, Y -71.294, Z 63.25, A 0, B 90, C 0, E1 0, E2 0, E3 0, E4 0} C_DIS
LIN {X 47.167, Y -73.305, Z 63.25, A 0, B 90, C 0, E1 0, E2 0, E3 0, E4 0} C_DIS
LIN {X 45.249, Y -75.058, Z 63.25, A 0, B 90, C 0, E1 0, E2 0, E3 0, E4 0} C_DIS
LIN {X 43.111, Y -76.535, Z 63.25, A 0, B 90, C 0, E1 0, E2 0, E3 0, E4 0} C_DIS
LIN {X 40.832, Y -77.786, Z 63.25, A 0, B 90, C 0, E1 0, E2 0, E3 0, E4 0} C_DIS
LIN {X 38.457, Y -78.842, Z 63.25, A 0, B 90, C 0, E1 0, E2 0, E3 0, E4 0} C_DIS
LIN {X 36.008, Y -79.715, Z 63.25, A 0, B 90, C 0, E1 0, E2 0, E3 0, E4 0} C_DIS
LIN {X 33.503, Y -80.413, Z 63.25, A 0, B 90, C 0, E1 0, E2 0, E3 0, E4 0} C_DIS
LIN {X 30.957, Y -80.938, Z 63.25, A 0, B 90, C 0, E1 0, E2 0, E3 0, E4 0} C_DIS
LIN {X 28.382, Y -81.295, Z 63.25, A 0, B 90, C 0, E1 0, E2 0, E3 0, E4 0} C_DIS
LIN {X 25.789, Y -81.491, Z 63.25, A 0, B 90, C 0, E1 0, E2 0, E3 0, E4 0} C_DIS
LIN {X 23.19, Y -81.538, Z 63.25, A 0, B 90, C 0, E1 0, E2 0, E3 0, E4 0} C_DIS
LIN {X 20.591, Y -81.454, Z 63.25, A 0, B 90, C 0, E1 0, E2 0, E3 0, E4 0} C_DIS
LIN {X 17.997, Y -81.27, Z 63.25, A 0, B 90, C 0, E1 0, E2 0, E3 0, E4 0} C_DIS
LIN {X 15.408, Y -81.03, Z 63.25, A 0, B 90, C 0, E1 0, E2 0, E3 0, E4 0} C_DIS
LIN {X 12.82, Y -80.773, Z 63.25, A 0, B 90, C 0, E1 0, E2 0, E3 0, E4 0} C_DIS
LIN {X 10.234, Y -80.496, Z 63.25, A 0, B 90, C 0, E1 0, E2 0, E3 0, E4 0} C_DIS
LIN {X 7.654, Y -80.174, Z 63.25, A 0, B 90, C 0, E1 0, E2 0, E3 0, E4 0} C_DIS
LIN {X 5.083, Y -79.784, Z 63.25, A 0, B 90, C 0, E1 0, E2 0, E3 0, E4 0} C_DIS
LIN {X 2.526, Y -79.315, Z 63.25, A 0, B 90, C 0, E1 0, E2 0, E3 0, E4 0} C_DIS
LIN {X 0, Y -78.741, Z 63.25, A 0, B 90, C 0, E1 0, E2 0, E3 0, E4 0} C_DIS
LIN {X -2.41, Y -77.914, Z 63.25, A 0, B 90, C 0, E1 0, E2 0, E3 0, E4 0} C_DIS
LIN {X -4.895, Y -77.148, Z 63.25, A 0, B 90, C 0, E1 0, E2 0, E3 0, E4 0} C_DIS
LIN {X -7.348, Y -76.286, Z 63.25, A 0, B 90, C 0, E1 0, E2 0, E3 0, E4 0} C_DIS
LIN {X -9.757, Y -75.306, Z 63.25, A 0, B 90, C 0, E1 0, E2 0, E3 0, E4 0} C_DIS
LIN {X -12.089, Y -74.159, Z 63.25, A 0, B 90, C 0, E1 0, E2 0, E3 0, E4 0} C_DIS
LIN {X -14.309, Y -72.805, Z 63.25, A 0, B 90, C 0, E1 0, E2 0, E3 0, E4 0} C_DIS
LIN {X -16.45, Y -71.33, Z 63.25, A 0, B 90, C 0, E1 0, E2 0, E3 0, E4 0} C_DIS
LIN {X -18.575, Y -69.832, Z 63.25, A 0, B 90, C 0, E1 0, E2 0, E3 0, E4 0} C_DIS
LIN {X -20.722, Y -68.364, Z 63.25, A 0, B 90, C 0, E1 0, E2 0, E3 0, E4 0} C_DIS
LIN {X -22.91, Y -66.959, Z 63.25, A 0, B 90, C 0, E1 0, E2 0, E3 0, E4 0} C_DIS
LIN {X -25.151, Y -65.64, Z 63.25, A 0, B 90, C 0, E1 0, E2 0, E3 0, E4 0} C_DIS
LIN {X -27.447, Y -64.42, Z 63.25, A 0, B 90, C 0, E1 0, E2 0, E3 0, E4 0} C_DIS
LIN {X -29.792, Y -63.298, Z 63.25, A 0, B 90, C 0, E1 0, E2 0, E3 0, E4 0} C_DIS
LIN {X -32.18, Y -62.268, Z 63.25, A 0, B 90, C 0, E1 0, E2 0, E3 0, E4 0} C_DIS
LIN {X -34.602, Y -61.322, Z 63.25, A 0, B 90, C 0, E1 0, E2 0, E3 0, E4 0} C_DIS
LIN {X -37.055, Y -60.459, Z 63.25, A 0, B 90, C 0, E1 0, E2 0, E3 0, E4 0} C_DIS
LIN {X -39.539, Y -59.691, Z 63.25, A 0, B 90, C 0, E1 0, E2 0, E3 0, E4 0} C_DIS
LIN {X -42.054, Y -59.031, Z 63.25, A 0, B 90, C 0, E1 0, E2 0, E3 0, E4 0} C_DIS
LIN {X -44.591, Y -58.46, Z 63.25, A 0, B 90, C 0, E1 0, E2 0, E3 0, E4 0} C_DIS
LIN {X -47.136, Y -57.929, Z 63.25, A 0, B 90, C 0, E1 0, E2 0, E3 0, E4 0} C_DIS
LIN {X -49.679, Y -57.385, Z 63.25, A 0, B 90, C 0, E1 0, E2 0, E3 0, E4 0} C_DIS
LIN {X -52.212, Y -56.796, Z 63.25, A 0, B 90, C 0, E1 0, E2 0, E3 0, E4 0} C_DIS
LIN {X -54.729, Y -56.142, Z 63.25, A 0, B 90, C 0, E1 0, E2 0, E3 0, E4 0} C_DIS
LIN {X -57.223, Y -55.408, Z 63.25, A 0, B 90, C 0, E1 0, E2 0, E3 0, E4 0} C_DIS
LIN {X -59.69, Y -54.587, Z 63.25, A 0, B 90, C 0, E1 0, E2 0, E3 0, E4 0} C_DIS
LIN {X -62.123, Y -53.668, Z 63.25, A 0, B 90, C 0, E1 0, E2 0, E3 0, E4 0} C_DIS
LIN {X -64.513, Y -52.645, Z 63.25, A 0, B 90, C 0, E1 0, E2 0, E3 0, E4 0} C_DIS
LIN {X -66.851, Y -51.507, Z 63.25, A 0, B 90, C 0, E1 0, E2 0, E3 0, E4 0} C_DIS
LIN {X -69.121, Y -50.239, Z 63.25, A 0, B 90, C 0, E1 0, E2 0, E3 0, E4 0} C_DIS
LIN {X -71.294, Y -48.812, Z 63.25, A 0, B 90, C 0, E1 0, E2 0, E3 0, E4 0} C_DIS
LIN {X -73.305, Y -47.167, Z 63.25, A 0, B 90, C 0, E1 0, E2 0, E3 0, E4 0} C_DIS
LIN {X -75.058, Y -45.249, Z 63.25, A 0, B 90, C 0, E1 0, E2 0, E3 0, E4 0} C_DIS
LIN {X -76.535, Y -43.111, Z 63.25, A 0, B 90, C 0, E1 0, E2 0, E3 0, E4 0} C_DIS
LIN {X -77.786, Y -40.832, Z 63.25, A 0, B 90, C 0, E1 0, E2 0, E3 0, E4 0} C_DIS
LIN {X -78.842, Y -38.457, Z 63.25, A 0, B 90, C 0, E1 0, E2 0, E3 0, E4 0} C_DIS
LIN {X -79.715, Y -36.008, Z 63.25, A 0, B 90, C 0, E1 0, E2 0, E3 0, E4 0} C_DIS
LIN {X -80.413, Y -33.503, Z 63.25, A 0, B 90, C 0, E1 0, E2 0, E3 0, E4 0} C_DIS
LIN {X -80.938, Y -30.957, Z 63.25, A 0, B 90, C 0, E1 0, E2 0, E3 0, E4 0} C_DIS
LIN {X -81.295, Y -28.382, Z 63.25, A 0, B 90, C 0, E1 0, E2 0, E3 0, E4 0} C_DIS
LIN {X -81.491, Y -25.789, Z 63.25, A 0, B 90, C 0, E1 0, E2 0, E3 0, E4 0} C_DIS
LIN {X -81.538, Y -23.19, Z 63.25, A 0, B 90, C 0, E1 0, E2 0, E3 0, E4 0} C_DIS
LIN {X -81.454, Y -20.591, Z 63.25, A 0, B 90, C 0, E1 0, E2 0, E3 0, E4 0} C_DIS
LIN {X -81.27, Y -17.997, Z 63.25, A 0, B 90, C 0, E1 0, E2 0, E3 0, E4 0} C_DIS
LIN {X -81.03, Y -15.408, Z 63.25, A 0, B 90, C 0, E1 0, E2 0, E3 0, E4 0} C_DIS
LIN {X -80.773, Y -12.82, Z 63.25, A 0, B 90, C 0, E1 0, E2 0, E3 0, E4 0} C_DIS
LIN {X -80.496, Y -10.234, Z 63.25, A 0, B 90, C 0, E1 0, E2 0, E3 0, E4 0} C_DIS
LIN {X -80.174, Y -7.654, Z 63.25, A 0, B 90, C 0, E1 0, E2 0, E3 0, E4 0} C_DIS
LIN {X -79.784, Y -5.083, Z 63.25, A 0, B 90, C 0, E1 0, E2 0, E3 0, E4 0} C_DIS
LIN {X -79.315, Y -2.526, Z 63.25, A 0, B 90, C 0, E1 0, E2 0, E3 0, E4 0} C_DIS
LIN {X -78.785, Y 0, Z 65.75, A 0, B 90, C 0, E1 0, E2 0, E3 0, E4 0} C_DIS
LIN {X -77.922, Y 2.402, Z 65.75, A 0, B 90, C 0, E1 0, E2 0, E3 0, E4 0} C_DIS
LIN {X -77.125, Y 4.887, Z 65.75, A 0, B 90, C 0, E1 0, E2 0, E3 0, E4 0} C_DIS
LIN {X -76.233, Y 7.339, Z 65.75, A 0, B 90, C 0, E1 0, E2 0, E3 0, E4 0} C_DIS
LIN {X -75.222, Y 9.745, Z 65.75, A 0, B 90, C 0, E1 0, E2 0, E3 0, E4 0} C_DIS
LIN {X -74.042, Y 12.072, Z 65.75, A 0, B 90, C 0, E1 0, E2 0, E3 0, E4 0} C_DIS
LIN {X -72.657, Y 14.283, Z 65.75, A 0, B 90, C 0, E1 0, E2 0, E3 0, E4 0} C_DIS
LIN {X -71.152, Y 16.415, Z 65.75, A 0, B 90, C 0, E1 0, E2 0, E3 0, E4 0} C_DIS
LIN {X -69.627, Y 18.533, Z 65.75, A 0, B 90, C 0, E1 0, E2 0, E3 0, E4 0} C_DIS
LIN {X -68.135, Y 20.674, Z 65.75, A 0, B 90, C 0, E1 0, E2 0, E3 0, E4 0} C_DIS
LIN {X -66.71, Y 22.861, Z 65.75, A 0, B 90, C 0, E1 0, E2 0, E3 0, E4 0} C_DIS
LIN {X -65.376, Y 25.103, Z 65.75, A 0, B 90, C 0, E1 0, E2 0, E3 0, E4 0} C_DIS
LIN {X -64.145, Y 27.404, Z 65.75, A 0, B 90, C 0, E1 0, E2 0, E3 0, E4 0} C_DIS
LIN {X -63.019, Y 29.759, Z 65.75, A 0, B 90, C 0, E1 0, E2 0, E3 0, E4 0} C_DIS
LIN {X -61.99, Y 32.157, Z 65.75, A 0, B 90, C 0, E1 0, E2 0, E3 0, E4 0} C_DIS
LIN {X -61.052, Y 34.592, Z 65.75, A 0, B 90, C 0, E1 0, E2 0, E3 0, E4 0} C_DIS
LIN {X -60.202, Y 37.06, Z 65.75, A 0, B 90, C 0, E1 0, E2 0, E3 0, E4 0} C_DIS
LIN {X -59.454, Y 39.56, Z 65.75, A 0, B 90, C 0, E1 0, E2 0, E3 0, E4 0} C_DIS
LIN {X -58.819, Y 42.091, Z 65.75, A 0, B 90, C 0, E1 0, E2 0, E3 0, E4 0} C_DIS
LIN {X -58.278, Y 44.644, Z 65.75, A 0, B 90, C 0, E1 0, E2 0, E3 0, E4 0} C_DIS
LIN {X -57.777, Y 47.205, Z 65.75, A 0, B 90, C 0, E1 0, E2 0, E3 0, E4 0} C_DIS
LIN {X -57.264, Y 49.764, Z 65.75, A 0, B 90, C 0, E1 0, E2 0, E3 0, E4 0} C_DIS
LIN {X -56.706, Y 52.314, Z 65.75, A 0, B 90, C 0, E1 0, E2 0, E3 0, E4 0} C_DIS
LIN {X -56.082, Y 54.848, Z 65.75, A 0, B 90, C 0, E1 0, E2 0, E3 0, E4 0} C_DIS
LIN {X -55.378, Y 57.361, Z 65.75, A 0, B 90, C 0, E1 0, E2 0, E3 0, E4 0} C_DIS
LIN {X -54.585, Y 59.847, Z 65.75, A 0, B 90, C 0, E1 0, E2 0, E3 0, E4 0} C_DIS
LIN {X -53.694, Y 62.3, Z 65.75, A 0, B 90, C 0, E1 0, E2 0, E3 0, E4 0} C_DIS
LIN {X -52.696, Y 64.711, Z 65.75, A 0, B 90, C 0, E1 0, E2 0, E3 0, E4 0} C_DIS
LIN {X -51.582, Y 67.071, Z 65.75, A 0, B 90, C 0, E1 0, E2 0, E3 0, E4 0} C_DIS
LIN {X -50.335, Y 69.363, Z 65.75, A 0, B 90, C 0, E1 0, E2 0, E3 0, E4 0} C_DIS
LIN {X -48.927, Y 71.559, Z 65.75, A 0, B 90, C 0, E1 0, E2 0, E3 0, E4 0} C_DIS
LIN {X -47.296, Y 73.594, Z 65.75, A 0, B 90, C 0, E1 0, E2 0, E3 0, E4 0} C_DIS
LIN {X -45.384, Y 75.367, Z 65.75, A 0, B 90, C 0, E1 0, E2 0, E3 0, E4 0} C_DIS
LIN {X -43.244, Y 76.858, Z 65.75, A 0, B 90, C 0, E1 0, E2 0, E3 0, E4 0} C_DIS
LIN {X -40.959, Y 78.118, Z 65.75, A 0, B 90, C 0, E1 0, E2 0, E3 0, E4 0} C_DIS
LIN {X -38.575, Y 79.178, Z 65.75, A 0, B 90, C 0, E1 0, E2 0, E3 0, E4 0} C_DIS
LIN {X -36.116, Y 80.051, Z 65.75, A 0, B 90, C 0, E1 0, E2 0, E3 0, E4 0} C_DIS
LIN {X -33.601, Y 80.744, Z 65.75, A 0, B 90, C 0, E1 0, E2 0, E3 0, E4 0} C_DIS
LIN {X -31.043, Y 81.261, Z 65.75, A 0, B 90, C 0, E1 0, E2 0, E3 0, E4 0} C_DIS
LIN {X -28.457, Y 81.606, Z 65.75, A 0, B 90, C 0, E1 0, E2 0, E3 0, E4 0} C_DIS
LIN {X -25.853, Y 81.787, Z 65.75, A 0, B 90, C 0, E1 0, E2 0, E3 0, E4 0} C_DIS
LIN {X -23.244, Y 81.815, Z 65.75, A 0, B 90, C 0, E1 0, E2 0, E3 0, E4 0} C_DIS
LIN {X -20.637, Y 81.709, Z 65.75, A 0, B 90, C 0, E1 0, E2 0, E3 0, E4 0} C_DIS
LIN {X -18.035, Y 81.501, Z 65.75, A 0, B 90, C 0, E1 0, E2 0, E3 0, E4 0} C_DIS
LIN {X -15.439, Y 81.236, Z 65.75, A 0, B 90, C 0, E1 0, E2 0, E3 0, E4 0} C_DIS
LIN {X -12.844, Y 80.953, Z 65.75, A 0, B 90, C 0, E1 0, E2 0, E3 0, E4 0} C_DIS
LIN {X -10.252, Y 80.65, Z 65.75, A 0, B 90, C 0, E1 0, E2 0, E3 0, E4 0} C_DIS
LIN {X -7.666, Y 80.301, Z 65.75, A 0, B 90, C 0, E1 0, E2 0, E3 0, E4 0} C_DIS
LIN {X -5.09, Y 79.883, Z 65.75, A 0, B 90, C 0, E1 0, E2 0, E3 0, E4 0} C_DIS
LIN {X -2.528, Y 79.387, Z 65.75, A 0, B 90, C 0, E1 0, E2 0, E3 0, E4 0} C_DIS
LIN {X 0, Y 78.785, Z 65.75, A 0, B 90, C 0, E1 0, E2 0, E3 0, E4 0} C_DIS
LIN {X 2.402, Y 77.922, Z 65.75, A 0, B 90, C 0, E1 0, E2 0, E3 0, E4 0} C_DIS
LIN {X 4.887, Y 77.125, Z 65.75, A 0, B 90, C 0, E1 0, E2 0, E3 0, E4 0} C_DIS
LIN {X 7.339, Y 76.233, Z 65.75, A 0, B 90, C 0, E1 0, E2 0, E3 0, E4 0} C_DIS
LIN {X 9.745, Y 75.222, Z 65.75, A 0, B 90, C 0, E1 0, E2 0, E3 0, E4 0} C_DIS
LIN {X 12.072, Y 74.042, Z 65.75, A 0, B 90, C 0, E1 0, E2 0, E3 0, E4 0} C_DIS
LIN {X 14.283, Y 72.657, Z 65.75, A 0, B 90, C 0, E1 0, E2 0, E3 0, E4 0} C_DIS
LIN {X 16.415, Y 71.152, Z 65.75, A 0, B 90, C 0, E1 0, E2 0, E3 0, E4 0} C_DIS
LIN {X 18.533, Y 69.627, Z 65.75, A 0, B 90, C 0, E1 0, E2 0, E3 0, E4 0} C_DIS
LIN {X 20.674, Y 68.135, Z 65.75, A 0, B 90, C 0, E1 0, E2 0, E3 0, E4 0} C_DIS
LIN {X 22.861, Y 66.71, Z 65.75, A 0, B 90, C 0, E1 0, E2 0, E3 0, E4 0} C_DIS
LIN {X 25.103, Y 65.376, Z 65.75, A 0, B 90, C 0, E1 0, E2 0, E3 0, E4 0} C_DIS
LIN {X 27.404, Y 64.145, Z 65.75, A 0, B 90, C 0, E1 0, E2 0, E3 0, E4 0} C_DIS
LIN {X 29.759, Y 63.019, Z 65.75, A 0, B 90, C 0, E1 0, E2 0, E3 0, E4 0} C_DIS
LIN {X 32.157, Y 61.99, Z 65.75, A 0, B 90, C 0, E1 0, E2 0, E3 0, E4 0} C_DIS
LIN {X 34.592, Y 61.052, Z 65.75, A 0, B 90, C 0, E1 0, E2 0, E3 0, E4 0} C_DIS
LIN {X 37.06, Y 60.202, Z 65.75, A 0, B 90, C 0, E1 0, E2 0, E3 0, E4 0} C_DIS
LIN {X 39.56, Y 59.454, Z 65.75, A 0, B 90, C 0, E1 0, E2 0, E3 0, E4 0} C_DIS
LIN {X 42.091, Y 58.819, Z 65.75, A 0, B 90, C 0, E1 0, E2 0, E3 0, E4 0} C_DIS
LIN {X 44.644, Y 58.278, Z 65.75, A 0, B 90, C 0, E1 0, E2 0, E3 0, E4 0} C_DIS
LIN {X 47.205, Y 57.777, Z 65.75, A 0, B 90, C 0, E1 0, E2 0, E3 0, E4 0} C_DIS
LIN {X 49.764, Y 57.264, Z 65.75, A 0, B 90, C 0, E1 0, E2 0, E3 0, E4 0} C_DIS
LIN {X 52.314, Y 56.706, Z 65.75, A 0, B 90, C 0, E1 0, E2 0, E3 0, E4 0} C_DIS
LIN {X 54.848, Y 56.082, Z 65.75, A 0, B 90, C 0, E1 0, E2 0, E3 0, E4 0} C_DIS
LIN {X 57.361, Y 55.378, Z 65.75, A 0, B 90, C 0, E1 0, E2 0, E3 0, E4 0} C_DIS
LIN {X 59.847, Y 54.585, Z 65.75, A 0, B 90, C 0, E1 0, E2 0, E3 0, E4 0} C_DIS
LIN {X 62.3, Y 53.694, Z 65.75, A 0, B 90, C 0, E1 0, E2 0, E3 0, E4 0} C_DIS
LIN {X 64.711, Y 52.696, Z 65.75, A 0, B 90, C 0, E1 0, E2 0, E3 0, E4 0} C_DIS
LIN {X 67.071, Y 51.582, Z 65.75, A 0, B 90, C 0, E1 0, E2 0, E3 0, E4 0} C_DIS
LIN {X 69.363, Y 50.335, Z 65.75, A 0, B 90, C 0, E1 0, E2 0, E3 0, E4 0} C_DIS
LIN {X 71.559, Y 48.927, Z 65.75, A 0, B 90, C 0, E1 0, E2 0, E3 0, E4 0} C_DIS
LIN {X 73.594, Y 47.296, Z 65.75, A 0, B 90, C 0, E1 0, E2 0, E3 0, E4 0} C_DIS
LIN {X 75.367, Y 45.384, Z 65.75, A 0, B 90, C 0, E1 0, E2 0, E3 0, E4 0} C_DIS
LIN {X 76.858, Y 43.244, Z 65.75, A 0, B 90, C 0, E1 0, E2 0, E3 0, E4 0} C_DIS
LIN {X 78.118, Y 40.959, Z 65.75, A 0, B 90, C 0, E1 0, E2 0, E3 0, E4 0} C_DIS
LIN {X 79.178, Y 38.575, Z 65.75, A 0, B 90, C 0, E1 0, E2 0, E3 0, E4 0} C_DIS
LIN {X 80.051, Y 36.116, Z 65.75, A 0, B 90, C 0, E1 0, E2 0, E3 0, E4 0} C_DIS
LIN {X 80.744, Y 33.601, Z 65.75, A 0, B 90, C 0, E1 0, E2 0, E3 0, E4 0} C_DIS
LIN {X 81.261, Y 31.043, Z 65.75, A 0, B 90, C 0, E1 0, E2 0, E3 0, E4 0} C_DIS
LIN {X 81.606, Y 28.457, Z 65.75, A 0, B 90, C 0, E1 0, E2 0, E3 0, E4 0} C_DIS
LIN {X 81.787, Y 25.853, Z 65.75, A 0, B 90, C 0, E1 0, E2 0, E3 0, E4 0} C_DIS
LIN {X 81.815, Y 23.244, Z 65.75, A 0, B 90, C 0, E1 0, E2 0, E3 0, E4 0} C_DIS
LIN {X 81.709, Y 20.637, Z 65.75, A 0, B 90, C 0, E1 0, E2 0, E3 0, E4 0} C_DIS
LIN {X 81.501, Y 18.035, Z 65.75, A 0, B 90, C 0, E1 0, E2 0, E3 0, E4 0} C_DIS
LIN {X 81.236, Y 15.439, Z 65.75, A 0, B 90, C 0, E1 0, E2 0, E3 0, E4 0} C_DIS
LIN {X 80.953, Y 12.844, Z 65.75, A 0, B 90, C 0, E1 0, E2 0, E3 0, E4 0} C_DIS
LIN {X 80.65, Y 10.252, Z 65.75, A 0, B 90, C 0, E1 0, E2 0, E3 0, E4 0} C_DIS
LIN {X 80.301, Y 7.666, Z 65.75, A 0, B 90, C 0, E1 0, E2 0, E3 0, E4 0} C_DIS
LIN {X 79.883, Y 5.09, Z 65.75, A 0, B 90, C 0, E1 0, E2 0, E3 0, E4 0} C_DIS
LIN {X 79.387, Y 2.528, Z 65.75, A 0, B 90, C 0, E1 0, E2 0, E3 0, E4 0} C_DIS
LIN {X 78.785, Y 0, Z 65.75, A 0, B 90, C 0, E1 0, E2 0, E3 0, E4 0} C_DIS
LIN {X 77.922, Y -2.402, Z 65.75, A 0, B 90, C 0, E1 0, E2 0, E3 0, E4 0} C_DIS
LIN {X 77.125, Y -4.887, Z 65.75, A 0, B 90, C 0, E1 0, E2 0, E3 0, E4 0} C_DIS
LIN {X 76.233, Y -7.339, Z 65.75, A 0, B 90, C 0, E1 0, E2 0, E3 0, E4 0} C_DIS
LIN {X 75.222, Y -9.745, Z 65.75, A 0, B 90, C 0, E1 0, E2 0, E3 0, E4 0} C_DIS
LIN {X 74.042, Y -12.072, Z 65.75, A 0, B 90, C 0, E1 0, E2 0, E3 0, E4 0} C_DIS
LIN {X 72.657, Y -14.283, Z 65.75, A 0, B 90, C 0, E1 0, E2 0, E3 0, E4 0} C_DIS
LIN {X 71.152, Y -16.415, Z 65.75, A 0, B 90, C 0, E1 0, E2 0, E3 0, E4 0} C_DIS
LIN {X 69.627, Y -18.533, Z 65.75, A 0, B 90, C 0, E1 0, E2 0, E3 0, E4 0} C_DIS
LIN {X 68.135, Y -20.674, Z 65.75, A 0, B 90, C 0, E1 0, E2 0, E3 0, E4 0} C_DIS
LIN {X 66.71, Y -22.861, Z 65.75, A 0, B 90, C 0, E1 0, E2 0, E3 0, E4 0} C_DIS
LIN {X 65.376, Y -25.103, Z 65.75, A 0, B 90, C 0, E1 0, E2 0, E3 0, E4 0} C_DIS
LIN {X 64.145, Y -27.404, Z 65.75, A 0, B 90, C 0, E1 0, E2 0, E3 0, E4 0} C_DIS
LIN {X 63.019, Y -29.759, Z 65.75, A 0, B 90, C 0, E1 0, E2 0, E3 0, E4 0} C_DIS
LIN {X 61.99, Y -32.157, Z 65.75, A 0, B 90, C 0, E1 0, E2 0, E3 0, E4 0} C_DIS
LIN {X 61.052, Y -34.592, Z 65.75, A 0, B 90, C 0, E1 0, E2 0, E3 0, E4 0} C_DIS
LIN {X 60.202, Y -37.06, Z 65.75, A 0, B 90, C 0, E1 0, E2 0, E3 0, E4 0} C_DIS
LIN {X 59.454, Y -39.56, Z 65.75, A 0, B 90, C 0, E1 0, E2 0, E3 0, E4 0} C_DIS
LIN {X 58.819, Y -42.091, Z 65.75, A 0, B 90, C 0, E1 0, E2 0, E3 0, E4 0} C_DIS
LIN {X 58.278, Y -44.644, Z 65.75, A 0, B 90, C 0, E1 0, E2 0, E3 0, E4 0} C_DIS
LIN {X 57.777, Y -47.205, Z 65.75, A 0, B 90, C 0, E1 0, E2 0, E3 0, E4 0} C_DIS
LIN {X 57.264, Y -49.764, Z 65.75, A 0, B 90, C 0, E1 0, E2 0, E3 0, E4 0} C_DIS
LIN {X 56.706, Y -52.314, Z 65.75, A 0, B 90, C 0, E1 0, E2 0, E3 0, E4 0} C_DIS
LIN {X 56.082, Y -54.848, Z 65.75, A 0, B 90, C 0, E1 0, E2 0, E3 0, E4 0} C_DIS
LIN {X 55.378, Y -57.361, Z 65.75, A 0, B 90, C 0, E1 0, E2 0, E3 0, E4 0} C_DIS
LIN {X 54.585, Y -59.847, Z 65.75, A 0, B 90, C 0, E1 0, E2 0, E3 0, E4 0} C_DIS
LIN {X 53.694, Y -62.3, Z 65.75, A 0, B 90, C 0, E1 0, E2 0, E3 0, E4 0} C_DIS
LIN {X 52.696, Y -64.711, Z 65.75, A 0, B 90, C 0, E1 0, E2 0, E3 0, E4 0} C_DIS
LIN {X 51.582, Y -67.071, Z 65.75, A 0, B 90, C 0, E1 0, E2 0, E3 0, E4 0} C_DIS
LIN {X 50.335, Y -69.363, Z 65.75, A 0, B 90, C 0, E1 0, E2 0, E3 0, E4 0} C_DIS
LIN {X 48.927, Y -71.559, Z 65.75, A 0, B 90, C 0, E1 0, E2 0, E3 0, E4 0} C_DIS
LIN {X 47.296, Y -73.594, Z 65.75, A 0, B 90, C 0, E1 0, E2 0, E3 0, E4 0} C_DIS
LIN {X 45.384, Y -75.367, Z 65.75, A 0, B 90, C 0, E1 0, E2 0, E3 0, E4 0} C_DIS
LIN {X 43.244, Y -76.858, Z 65.75, A 0, B 90, C 0, E1 0, E2 0, E3 0, E4 0} C_DIS
LIN {X 40.959, Y -78.118, Z 65.75, A 0, B 90, C 0, E1 0, E2 0, E3 0, E4 0} C_DIS
LIN {X 38.575, Y -79.178, Z 65.75, A 0, B 90, C 0, E1 0, E2 0, E3 0, E4 0} C_DIS
LIN {X 36.116, Y -80.051, Z 65.75, A 0, B 90, C 0, E1 0, E2 0, E3 0, E4 0} C_DIS
LIN {X 33.601, Y -80.744, Z 65.75, A 0, B 90, C 0, E1 0, E2 0, E3 0, E4 0} C_DIS
LIN {X 31.043, Y -81.261, Z 65.75, A 0, B 90, C 0, E1 0, E2 0, E3 0, E4 0} C_DIS
LIN {X 28.457, Y -81.606, Z 65.75, A 0, B 90, C 0, E1 0, E2 0, E3 0, E4 0} C_DIS
LIN {X 25.853, Y -81.787, Z 65.75, A 0, B 90, C 0, E1 0, E2 0, E3 0, E4 0} C_DIS
LIN {X 23.244, Y -81.815, Z 65.75, A 0, B 90, C 0, E1 0, E2 0, E3 0, E4 0} C_DIS
LIN {X 20.637, Y -81.709, Z 65.75, A 0, B 90, C 0, E1 0, E2 0, E3 0, E4 0} C_DIS
LIN {X 18.035, Y -81.501, Z 65.75, A 0, B 90, C 0, E1 0, E2 0, E3 0, E4 0} C_DIS
LIN {X 15.439, Y -81.236, Z 65.75, A 0, B 90, C 0, E1 0, E2 0, E3 0, E4 0} C_DIS
LIN {X 12.844, Y -80.953, Z 65.75, A 0, B 90, C 0, E1 0, E2 0, E3 0, E4 0} C_DIS
LIN {X 10.252, Y -80.65, Z 65.75, A 0, B 90, C 0, E1 0, E2 0, E3 0, E4 0} C_DIS
LIN {X 7.666, Y -80.301, Z 65.75, A 0, B 90, C 0, E1 0, E2 0, E3 0, E4 0} C_DIS
LIN {X 5.09, Y -79.883, Z 65.75, A 0, B 90, C 0, E1 0, E2 0, E3 0, E4 0} C_DIS
LIN {X 2.528, Y -79.387, Z 65.75, A 0, B 90, C 0, E1 0, E2 0, E3 0, E4 0} C_DIS
LIN {X 0, Y -78.785, Z 65.75, A 0, B 90, C 0, E1 0, E2 0, E3 0, E4 0} C_DIS
LIN {X -2.402, Y -77.922, Z 65.75, A 0, B 90, C 0, E1 0, E2 0, E3 0, E4 0} C_DIS
LIN {X -4.887, Y -77.125, Z 65.75, A 0, B 90, C 0, E1 0, E2 0, E3 0, E4 0} C_DIS
LIN {X -7.339, Y -76.233, Z 65.75, A 0, B 90, C 0, E1 0, E2 0, E3 0, E4 0} C_DIS
LIN {X -9.745, Y -75.222, Z 65.75, A 0, B 90, C 0, E1 0, E2 0, E3 0, E4 0} C_DIS
LIN {X -12.072, Y -74.042, Z 65.75, A 0, B 90, C 0, E1 0, E2 0, E3 0, E4 0} C_DIS
LIN {X -14.283, Y -72.657, Z 65.75, A 0, B 90, C 0, E1 0, E2 0, E3 0, E4 0} C_DIS
LIN {X -16.415, Y -71.152, Z 65.75, A 0, B 90, C 0, E1 0, E2 0, E3 0, E4 0} C_DIS
LIN {X -18.533, Y -69.627, Z 65.75, A 0, B 90, C 0, E1 0, E2 0, E3 0, E4 0} C_DIS
LIN {X -20.674, Y -68.135, Z 65.75, A 0, B 90, C 0, E1 0, E2 0, E3 0, E4 0} C_DIS
LIN {X -22.861, Y -66.71, Z 65.75, A 0, B 90, C 0, E1 0, E2 0, E3 0, E4 0} C_DIS
LIN {X -25.103, Y -65.376, Z 65.75, A 0, B 90, C 0, E1 0, E2 0, E3 0, E4 0} C_DIS
LIN {X -27.404, Y -64.145, Z 65.75, A 0, B 90, C 0, E1 0, E2 0, E3 0, E4 0} C_DIS
LIN {X -29.759, Y -63.019, Z 65.75, A 0, B 90, C 0, E1 0, E2 0, E3 0, E4 0} C_DIS
LIN {X -32.157, Y -61.99, Z 65.75, A 0, B 90, C 0, E1 0, E2 0, E3 0, E4 0} C_DIS
LIN {X -34.592, Y -61.052, Z 65.75, A 0, B 90, C 0, E1 0, E2 0, E3 0, E4 0} C_DIS
LIN {X -37.06, Y -60.202, Z 65.75, A 0, B 90, C 0, E1 0, E2 0, E3 0, E4 0} C_DIS
LIN {X -39.56, Y -59.454, Z 65.75, A 0, B 90, C 0, E1 0, E2 0, E3 0, E4 0} C_DIS
LIN {X -42.091, Y -58.819, Z 65.75, A 0, B 90, C 0, E1 0, E2 0, E3 0, E4 0} C_DIS
LIN {X -44.644, Y -58.278, Z 65.75, A 0, B 90, C 0, E1 0, E2 0, E3 0, E4 0} C_DIS
LIN {X -47.205, Y -57.777, Z 65.75, A 0, B 90, C 0, E1 0, E2 0, E3 0, E4 0} C_DIS
LIN {X -49.764, Y -57.264, Z 65.75, A 0, B 90, C 0, E1 0, E2 0, E3 0, E4 0} C_DIS
LIN {X -52.314, Y -56.706, Z 65.75, A 0, B 90, C 0, E1 0, E2 0, E3 0, E4 0} C_DIS
LIN {X -54.848, Y -56.082, Z 65.75, A 0, B 90, C 0, E1 0, E2 0, E3 0, E4 0} C_DIS
LIN {X -57.361, Y -55.378, Z 65.75, A 0, B 90, C 0, E1 0, E2 0, E3 0, E4 0} C_DIS
LIN {X -59.847, Y -54.585, Z 65.75, A 0, B 90, C 0, E1 0, E2 0, E3 0, E4 0} C_DIS
LIN {X -62.3, Y -53.694, Z 65.75, A 0, B 90, C 0, E1 0, E2 0, E3 0, E4 0} C_DIS
LIN {X -64.711, Y -52.696, Z 65.75, A 0, B 90, C 0, E1 0, E2 0, E3 0, E4 0} C_DIS
LIN {X -67.071, Y -51.582, Z 65.75, A 0, B 90, C 0, E1 0, E2 0, E3 0, E4 0} C_DIS
LIN {X -69.363, Y -50.335, Z 65.75, A 0, B 90, C 0, E1 0, E2 0, E3 0, E4 0} C_DIS
LIN {X -71.559, Y -48.927, Z 65.75, A 0, B 90, C 0, E1 0, E2 0, E3 0, E4 0} C_DIS
LIN {X -73.594, Y -47.296, Z 65.75, A 0, B 90, C 0, E1 0, E2 0, E3 0, E4 0} C_DIS
LIN {X -75.367, Y -45.384, Z 65.75, A 0, B 90, C 0, E1 0, E2 0, E3 0, E4 0} C_DIS
LIN {X -76.858, Y -43.244, Z 65.75, A 0, B 90, C 0, E1 0, E2 0, E3 0, E4 0} C_DIS
LIN {X -78.118, Y -40.959, Z 65.75, A 0, B 90, C 0, E1 0, E2 0, E3 0, E4 0} C_DIS
LIN {X -79.178, Y -38.575, Z 65.75, A 0, B 90, C 0, E1 0, E2 0, E3 0, E4 0} C_DIS
LIN {X -80.051, Y -36.116, Z 65.75, A 0, B 90, C 0, E1 0, E2 0, E3 0, E4 0} C_DIS
LIN {X -80.744, Y -33.601, Z 65.75, A 0, B 90, C 0, E1 0, E2 0, E3 0, E4 0} C_DIS
LIN {X -81.261, Y -31.043, Z 65.75, A 0, B 90, C 0, E1 0, E2 0, E3 0, E4 0} C_DIS
LIN {X -81.606, Y -28.457, Z 65.75, A 0, B 90, C 0, E1 0, E2 0, E3 0, E4 0} C_DIS
LIN {X -81.787, Y -25.853, Z 65.75, A 0, B 90, C 0, E1 0, E2 0, E3 0, E4 0} C_DIS
LIN {X -81.815, Y -23.244, Z 65.75, A 0, B 90, C 0, E1 0, E2 0, E3 0, E4 0} C_DIS
LIN {X -81.709, Y -20.637, Z 65.75, A 0, B 90, C 0, E1 0, E2 0, E3 0, E4 0} C_DIS
LIN {X -81.501, Y -18.035, Z 65.75, A 0, B 90, C 0, E1 0, E2 0, E3 0, E4 0} C_DIS
LIN {X -81.236, Y -15.439, Z 65.75, A 0, B 90, C 0, E1 0, E2 0, E3 0, E4 0} C_DIS
LIN {X -80.953, Y -12.844, Z 65.75, A 0, B 90, C 0, E1 0, E2 0, E3 0, E4 0} C_DIS
LIN {X -80.65, Y -10.252, Z 65.75, A 0, B 90, C 0, E1 0, E2 0, E3 0, E4 0} C_DIS
LIN {X -80.301, Y -7.666, Z 65.75, A 0, B 90, C 0, E1 0, E2 0, E3 0, E4 0} C_DIS
LIN {X -79.883, Y -5.09, Z 65.75, A 0, B 90, C 0, E1 0, E2 0, E3 0, E4 0} C_DIS
LIN {X -79.387, Y -2.528, Z 65.75, A 0, B 90, C 0, E1 0, E2 0, E3 0, E4 0} C_DIS
LIN {X -78.837, Y 0, Z 68.25, A 0, B 90, C 0, E1 0, E2 0, E3 0, E4 0} C_DIS
LIN {X -77.939, Y 2.393, Z 68.25, A 0, B 90, C 0, E1 0, E2 0, E3 0, E4 0} C_DIS
LIN {X -77.112, Y 4.878, Z 68.25, A 0, B 90, C 0, E1 0, E2 0, E3 0, E4 0} C_DIS
LIN {X -76.189, Y 7.33, Z 68.25, A 0, B 90, C 0, E1 0, E2 0, E3 0, E4 0} C_DIS
LIN {X -75.147, Y 9.733, Z 68.25, A 0, B 90, C 0, E1 0, E2 0, E3 0, E4 0} C_DIS
LIN {X -73.937, Y 12.055, Z 68.25, A 0, B 90, C 0, E1 0, E2 0, E3 0, E4 0} C_DIS
LIN {X -72.521, Y 14.258, Z 68.25, A 0, B 90, C 0, E1 0, E2 0, E3 0, E4 0} C_DIS
LIN {X -70.987, Y 16.382, Z 68.25, A 0, B 90, C 0, E1 0, E2 0, E3 0, E4 0} C_DIS
LIN {X -69.436, Y 18.493, Z 68.25, A 0, B 90, C 0, E1 0, E2 0, E3 0, E4 0} C_DIS
LIN {X -67.922, Y 20.63, Z 68.25, A 0, B 90, C 0, E1 0, E2 0, E3 0, E4 0} C_DIS
LIN {X -66.477, Y 22.815, Z 68.25, A 0, B 90, C 0, E1 0, E2 0, E3 0, E4 0} C_DIS
LIN {X -65.128, Y 25.06, Z 68.25, A 0, B 90, C 0, E1 0, E2 0, E3 0, E4 0} C_DIS
LIN {X -63.887, Y 27.367, Z 68.25, A 0, B 90, C 0, E1 0, E2 0, E3 0, E4 0} C_DIS
LIN {X -62.757, Y 29.73, Z 68.25, A 0, B 90, C 0, E1 0, E2 0, E3 0, E4 0} C_DIS
LIN {X -61.731, Y 32.14, Z 68.25, A 0, B 90, C 0, E1 0, E2 0, E3 0, E4 0} C_DIS
LIN {X -60.8, Y 34.588, Z 68.25, A 0, B 90, C 0, E1 0, E2 0, E3 0, E4 0} C_DIS
LIN {X -59.964, Y 37.071, Z 68.25, A 0, B 90, C 0, E1 0, E2 0, E3 0, E4 0} C_DIS
LIN {X -59.235, Y 39.586, Z 68.25, A 0, B 90, C 0, E1 0, E2 0, E3 0, E4 0} C_DIS
LIN {X -58.624, Y 42.133, Z 68.25, A 0, B 90, C 0, E1 0, E2 0, E3 0, E4 0} C_DIS
LIN {X -58.111, Y 44.702, Z 68.25, A 0, B 90, C 0, E1 0, E2 0, E3 0, E4 0} C_DIS
LIN {X -57.639, Y 47.279, Z 68.25, A 0, B 90, C 0, E1 0, E2 0, E3 0, E4 0} C_DIS
LIN {X -57.157, Y 49.853, Z 68.25, A 0, B 90, C 0, E1 0, E2 0, E3 0, E4 0} C_DIS
LIN {X -56.628, Y 52.419, Z 68.25, A 0, B 90, C 0, E1 0, E2 0, E3 0, E4 0} C_DIS
LIN {X -56.033, Y 54.97, Z 68.25, A 0, B 90, C 0, E1 0, E2 0, E3 0, E4 0} C_DIS
LIN {X -55.357, Y 57.501, Z 68.25, A 0, B 90, C 0, E1 0, E2 0, E3 0, E4 0} C_DIS
LIN {X -54.591, Y 60.005, Z 68.25, A 0, B 90, C 0, E1 0, E2 0, E3 0, E4 0} C_DIS
LIN {X -53.725, Y 62.478, Z 68.25, A 0, B 90, C 0, E1 0, E2 0, E3 0, E4 0} C_DIS
LIN {X -52.752, Y 64.909, Z 68.25, A 0, B 90, C 0, E1 0, E2 0, E3 0, E4 0} C_DIS
LIN {X -51.66, Y 67.29, Z 68.25, A 0, B 90, C 0, E1 0, E2 0, E3 0, E4 0} C_DIS
LIN {X -50.433, Y 69.604, Z 68.25, A 0, B 90, C 0, E1 0, E2 0, E3 0, E4 0} C_DIS
LIN {X -49.043, Y 71.823, Z 68.25, A 0, B 90, C 0, E1 0, E2 0, E3 0, E4 0} C_DIS
LIN {X -47.425, Y 73.881, Z 68.25, A 0, B 90, C 0, E1 0, E2 0, E3 0, E4 0} C_DIS
LIN {X -45.519, Y 75.674, Z 68.25, A 0, B 90, C 0, E1 0, E2 0, E3 0, E4 0} C_DIS
LIN {X -43.377, Y 77.18, Z 68.25, A 0, B 90, C 0, E1 0, E2 0, E3 0, E4 0} C_DIS
LIN {X -41.086, Y 78.448, Z 68.25, A 0, B 90, C 0, E1 0, E2 0, E3 0, E4 0} C_DIS
LIN {X -38.694, Y 79.513, Z 68.25, A 0, B 90, C 0, E1 0, E2 0, E3 0, E4 0} C_DIS
LIN {X -36.225, Y 80.387, Z 68.25, A 0, B 90, C 0, E1 0, E2 0, E3 0, E4 0} C_DIS
LIN {X -33.698, Y 81.076, Z 68.25, A 0, B 90, C 0, E1 0, E2 0, E3 0, E4 0} C_DIS
LIN {X -31.129, Y 81.585, Z 68.25, A 0, B 90, C 0, E1 0, E2 0, E3 0, E4 0} C_DIS
LIN {X -28.532, Y 81.919, Z 68.25, A 0, B 90, C 0, E1 0, E2 0, E3 0, E4 0} C_DIS
LIN {X -25.918, Y 82.086, Z 68.25, A 0, B 90, C 0, E1 0, E2 0, E3 0, E4 0} C_DIS
LIN {X -23.299, Y 82.097, Z 68.25, A 0, B 90, C 0, E1 0, E2 0, E3 0, E4 0} C_DIS
LIN {X -20.682, Y 81.971, Z 68.25, A 0, B 90, C 0, E1 0, E2 0, E3 0, E4 0} C_DIS
LIN {X -18.073, Y 81.74, Z 68.25, A 0, B 90, C 0, E1 0, E2 0, E3 0, E4 0} C_DIS
LIN {X -15.47, Y 81.45, Z 68.25, A 0, B 90, C 0, E1 0, E2 0, E3 0, E4 0} C_DIS
LIN {X -12.869, Y 81.141, Z 68.25, A 0, B 90, C 0, E1 0, E2 0, E3 0, E4 0} C_DIS
LIN {X -10.27, Y 80.813, Z 68.25, A 0, B 90, C 0, E1 0, E2 0, E3 0, E4 0} C_DIS
LIN {X -7.677, Y 80.437, Z 68.25, A 0, B 90, C 0, E1 0, E2 0, E3 0, E4 0} C_DIS
LIN {X -5.096, Y 79.992, Z 68.25, A 0, B 90, C 0, E1 0, E2 0, E3 0, E4 0} C_DIS
LIN {X -2.53, Y 79.468, Z 68.25, A 0, B 90, C 0, E1 0, E2 0, E3 0, E4 0} C_DIS
LIN {X 0, Y 78.837, Z 68.25, A 0, B 90, C 0, E1 0, E2 0, E3 0, E4 0} C_DIS
LIN {X 2.393, Y 77.939, Z 68.25, A 0, B 90, C 0, E1 0, E2 0, E3 0, E4 0} C_DIS
LIN {X 4.878, Y 77.112, Z 68.25, A 0, B 90, C 0, E1 0, E2 0, E3 0, E4 0} C_DIS
LIN {X 7.33, Y 76.189, Z 68.25, A 0, B 90, C 0, E1 0, E2 0, E3 0, E4 0} C_DIS
LIN {X 9.733, Y 75.147, Z 68.25, A 0, B 90, C 0, E1 0, E2 0, E3 0, E4 0} C_DIS
LIN {X 12.055, Y 73.937, Z 68.25, A 0, B 90, C 0, E1 0, E2 0, E3 0, E4 0} C_DIS
LIN {X 14.258, Y 72.521, Z 68.25, A 0, B 90, C 0, E1 0, E2 0, E3 0, E4 0} C_DIS
LIN {X 16.382, Y 70.987, Z 68.25, A 0, B 90, C 0, E1 0, E2 0, E3 0, E4 0} C_DIS
LIN {X 18.493, Y 69.436, Z 68.25, A 0, B 90, C 0, E1 0, E2 0, E3 0, E4 0} C_DIS
LIN {X 20.63, Y 67.922, Z 68.25, A 0, B 90, C 0, E1 0, E2 0, E3 0, E4 0} C_DIS
LIN {X 22.815, Y 66.477, Z 68.25, A 0, B 90, C 0, E1 0, E2 0, E3 0, E4 0} C_DIS
LIN {X 25.06, Y 65.128, Z 68.25, A 0, B 90, C 0, E1 0, E2 0, E3 0, E4 0} C_DIS
LIN {X 27.367, Y 63.887, Z 68.25, A 0, B 90, C 0, E1 0, E2 0, E3 0, E4 0} C_DIS
LIN {X 29.73, Y 62.757, Z 68.25, A 0, B 90, C 0, E1 0, E2 0, E3 0, E4 0} C_DIS
LIN {X 32.14, Y 61.731, Z 68.25, A 0, B 90, C 0, E1 0, E2 0, E3 0, E4 0} C_DIS
LIN {X 34.588, Y 60.8, Z 68.25, A 0, B 90, C 0, E1 0, E2 0, E3 0, E4 0} C_DIS
LIN {X 37.071, Y 59.964, Z 68.25, A 0, B 90, C 0, E1 0, E2 0, E3 0, E4 0} C_DIS
LIN {X 39.586, Y 59.235, Z 68.25, A 0, B 90, C 0, E1 0, E2 0, E3 0, E4 0} C_DIS
LIN {X 42.133, Y 58.624, Z 68.25, A 0, B 90, C 0, E1 0, E2 0, E3 0, E4 0} C_DIS
LIN {X 44.702, Y 58.111, Z 68.25, A 0, B 90, C 0, E1 0, E2 0, E3 0, E4 0} C_DIS
LIN {X 47.279, Y 57.639, Z 68.25, A 0, B 90, C 0, E1 0, E2 0, E3 0, E4 0} C_DIS
LIN {X 49.853, Y 57.157, Z 68.25, A 0, B 90, C 0, E1 0, E2 0, E3 0, E4 0} C_DIS
LIN {X 52.419, Y 56.628, Z 68.25, A 0, B 90, C 0, E1 0, E2 0, E3 0, E4 0} C_DIS
